60:
	AllGohomeTon[2].IN:=FALSE;
	Mach_Control.Ca_b.Ca_BeltGohomeHMI:=FALSE;
	Mach_Control.TJ_b.TJIniti_Hbtn:=FALSE;
	AllGohomeStep:=70;

70:
	AllGohomeTon[3].IN:=TRUE;
	IF AllGohomeTon[3].Q AND Mach_Control.Ca_b.Ca_BeltGohomeDone AND Mach_Control.TJ_b.TJIniti_Done THEN
	AllGohomeStep:=80;	
	END_IF	
80:
AllGohomeTon[3].IN:=FALSE;
AllGohomeStep:=888;	
END_CASE
END_ACTION

ACTION An_Alarm:


//报警时间
An_AlarmTon[1](IN:= , PT:=T#80MS , Q=> , ET=> );//正极送片搬运升降有真空信号，无极片报警延时
An_AlarmTon[2](IN:= , PT:=T#80MS , Q=> , ET=> );//正极送片搬运升降有极片，无真空信号报警延时
An_AlarmTon[3](IN:= , PT:=T#150MS , Q=> , ET=> );//正极叠台搬运升降有真空信号，无极片报警延时
An_AlarmTon[4](IN:= , PT:=T#80MS , Q=> , ET=> );//正极叠台搬运升降有极片，无真空信号报警延时
An_AlarmTon[5](IN:= , PT:=T#80MS , Q=> , ET=> );//正极纠偏平台有真空信号，无极片报警延时
An_AlarmTon[6](IN:= , PT:=T#150MS , Q=> , ET=> );//正极纠偏平台有极片，无真空信号报警延时
An_AlarmTon[7](IN:= , PT:=T#80MS , Q=> , ET=> );//正极纠偏平台连续NG
An_AlarmTon[8](IN:= , PT:=T#80MS , Q=> , ET=> );
An_AlarmTon[9](IN:= , PT:=T#300MS , Q=> , ET=> );
An_AlarmTon[10](IN:= , PT:=T#400MS , Q=> , ET=> );//
An_AlarmTon[11](IN:= , PT:=T#300MS , Q=> , ET=> );//正极极片对齐度检测返回结果超时
An_AlarmTon[12](IN:= , PT:=T#400MS , Q=> , ET=> );//正极CCD纠偏平台检测返回结果超时
An_AlarmTon[13](IN:=AnCCDMark , PT:=T#50MS , Q=> , ET=> );//正极CCD纠偏平台检测返回结果超时

An_AlarmTon[15](IN:= , PT:=T#50MS , Q=> , ET=> );//正极CCD纠偏平台检测返回结果超时
An_AlarmTon[16](IN:= , PT:=T#50MS , Q=> , ET=> );//正极CCD纠偏平台检测返回结果超时
An_AlarmTon[17](IN:=NOT Mach_Control.se.AnNGboxsensor , PT:=T#5S , Q=> , ET=> );//正极NG料盒料满

rAnUse[2](CLK:=Mach_Control.An_b.An_CCDStart AND NOT   Mach_Control.An_b.Demarcateing , Q=> );
rAnUse[3](CLK:=Par.stDT_date.An_Rectifydev_Btn , Q=> );
rAnUse[4](CLK:=arrCyCtrl[arrCyNo.ElectValveName.AnCarryingVacuum].Io.DOStatus1 , Q=> );  
rAnUse[5](CLK:= NOT arrCyCtrl[arrCyNo.ElectValveName.AnDTCarryingVacuum].Io.DOStatus1 , Q=> );

//Mach_Control.An_b.Error[1] :=TRUE;//正极送片搬运升降有真空信号，无极片报警
//Mach_Control.An_b.Error[2] :=TRUE;//正极送片搬运升降有极片，无真空信号报警
//Mach_Control.An_b.Error[3]:=TRUE;//正极叠台搬运升降在叠片过程中真空报警，请检查叠台是否掉片
//Mach_Control.An_b.Error[4] :=TRUE;//正极叠台搬运升降有极片，无真空信号报警
//Mach_Control.An_b.Error[5]:=TRUE;//正极纠偏平台有真空信号，无极片报警
//Mach_Control.An_b.Error[6]:=TRUE;//正极纠偏平台有极片，无真空信号报警
//Mach_Control.An_b.Error[7]:=TRUE;//纠偏CCD拍照完成IO信号未给出
//Mach_Control.An_b.Error[8]  ;//CCD标定NG
//Mach_Control.An_b.Error[9]  ;
//Mach_Control.An_b.Error[10]  ;
//Mach_Control.An_b.Error[11]:=TRUE;//正极有凸轮耦合报警
//Mach_Control.An_b.Error[12]:=TRUE;//正极NG收纳盒满料报警
//Mach_Control.An_b.Error[13];
//Mach_Control.An_b.Error[14]:=TRUE;//正极防撞感应信号报警
//Mach_Control.An_b.Error[15]
//Mach_Control.An_b.Error[16]
//Mach_Control.An_b.Error[17]
//Mach_Control.An_b.Error[18] :=TRUE;//正极CCD纠偏平台检测返回结果超时
// Mach_Control.An_b.Error[19]:=TRUE;//正极回原点超时报警
// Mach_Control.An_b.Error[20];
//Mach_Control.An_b.Error[21]:=TRUE;//正极纠偏平台连续NG
//Mach_Control.An_b.Error[22]:=TRUE;//正极叠台搬运升降真空报警，电芯上有片，请拿掉
//Mach_Control.An_b.Error[23]:=TRUE;//正极叠台搬运升降真空报警，电芯上无掉片
//Mach_Control.An_b.Error[24] ////正极纠偏平台NG片未排掉报警，请拿掉
//Mach_Control.An_b.Error[25] ////正极极片对齐度检测返回结果超时
//Mach_Control.An_b.Error[26] ////正极搬运防撞软限位报警
//Mach_Control.An_b.Error[27]//    //正极极片对齐度检测返回结果无片报警
//Mach_Control.An_b.Error[28]//正极叠片完空叠隔膜时，正极叠片搬运机械手真空有信号、标记有极片报警,请拿掉极片
//Mach_Control.An_b.Error[29]:=TRUE;		//正极初始化时正极叠片搬运升降吸盘有真空报警
//Mach_Control.An_b.Error[30]:=TRUE;		//正极初始化时正极送片搬运升降吸盘有真空报警	

//Mach_Control.An_b.Error[32]:=TRUE;//正极送片搬运在叠片过程中真空报警
//Mach_Control.An_b.Error[33]:=FALSE;//纠偏平台有片，请拿走
//Mach_Control.An_b.Error[34]:=FALSE;//正极叠台搬运平移取片时真空报警,请确认纠偏台是否掉片
//Mach_Control.An_b.Error[35]:=TRUE;//正极纠偏台NG料盒料满报警
//Mach_Control.An_b.Error[36]:=TRUE;//正极纠偏纠偏CCD返回结果超时
//Mach_Control.An_b.Error[37]:=TRUE;//正极叠台搬运升降有真空信号，无极片报警
//Mach_Control.An_b.Error[38] :=TRUE;//正极叠台搬运升降有极耳无真空报警
//Mach_Control.An_b.Error[39] :=TRUE;//正极叠台搬运升降有极耳无真空报警
//Mach_Control.An_b.Error[40] S=AnOverNGcount>=3;//正极单张踢废连续NG
//Mach_Control.An_b.Error[41] :=TRUE;//正极机械手初始化时，叠台搬运升降不在避让位
Mach_Control.An_b.Error[40] S=AnOverNGcount>=3;//正极单张踢废连续NG

//NG料盒料满报警
	IF (*Par.stDT_date.An_Rectifydev_JS>=Par.stDT_date.An_Rectifydev_NGSet OR*) An_AlarmTon[17].Q THEN
		Mach_Control.An_b.Error[35]:=TRUE;//负极纠偏台NG料盒料满报警
	ELSE
		Mach_Control.An_b.Error[35]:=FALSE;//负极纠偏台NG料盒料满报警
	END_IF
	IF rAnUse[3].Q THEN
		Par.stDT_date.An_Rectifydev_JS:=0;
	END_IF



//正极初始化时有真空报警	
	IF Mach_Control.An_b.An_GohomeHMI THEN
		IF arrCyCtrl[arrCyNo.ElectValveName.AnDTCarryingVacuum].Status.ONState  THEN    
			Mach_Control.An_b.Error[29]:=TRUE;		//正极初始化时正极叠片搬运升降吸盘有真空报警
		END_IF
		IF arrCyCtrl[arrCyNo.ElectValveName.	AnCarryingVacuum	].Status.ONState THEN	
			Mach_Control.An_b.Error[30]:=TRUE;		//正极初始化时正极送片搬运升降吸盘有真空报警	
		END_IF		 
	END_IF	
(*
//正极送片搬运升降真空信号与有无极片标记不一致报警
An_AlarmTon[1].IN:=arrCyCtrl[arrCyNo.ElectValveName.AnCarryingVacuum].Io.DIOnSwitch AND NOT Mach_Control.An_b.An_CarryingFalg 
	AND NOT Mach_Control.U.EmptyRunMode AND NOT Mach_Control.An_b.Error[2]  AND NOT Blueflaging AND Mach_Control.U.DT_iMode=1;
		IF  An_AlarmTon[1].Q THEN
				Mach_Control.An_b.Error[1] :=TRUE;//正极送片搬运升降有真空信号，无极片报警
		END_IF
*)
//正极送片搬运升降有极片，无真空信号报警------取片过程中真空报警判断
An_AlarmTon[2].IN:=NOT arrCyCtrl[arrCyNo.ElectValveName.AnCarryingVacuum].Io.DIOnSwitch AND  Mach_Control.An_b.An_CarryingFalg  AND
	 arrAxisCtrl[AxiseNo.AxisName.AnCarryingUpDown].Status.fActPos<=(arrAxisPar[AxiseNo.AxisName.AnCarryingUpDown].arrTargetPoint[2]-5) 
	AND arrAxisCtrl[AxiseNo.AxisName.AnCarryingLine].Status.NoMoving AND NOT Mach_Control.U.EmptyRunMode ;
	IF  An_AlarmTon[2].Q THEN
			Mach_Control.An_b.Error[2] :=TRUE;//正极送片搬运升降有极片，无真空信号报警
			(*
			Mach_Control.An_b.An_CarryingFalg:=FALSE;
			arrCyCtrl[arrCyNo.ElectValveName.AnCarryingVacuum].Cmd.bOFF:=TRUE;//正极搬运升降取料真空关
			arrCyCtrl[arrCyNo.ElectValveName.AnCarryingVacuum].Cmd.bON:=FALSE;//正极搬运升降取料真空关
			arrCyCtrl[arrCyNo.ElectValveName.AnCarryingVacuumBark].Cmd.bON:=TRUE;//正极搬运升降取料破真空开
			arrCyCtrl[arrCyNo.ElectValveName.AnCarryingVacuumBark].Cmd.bOFF:=FALSE;//正极搬运升降取料破真空开
			*)
	END_IF
IF 	Mach_Control.An_b.Error[2]AND arrCyCtrl[arrCyNo.ElectValveName.AnCarryingVacuum].Io.DIOnSwitch AND  rAn_AlarmRest.Q  THEN
	Mach_Control.An_b.Error[2] :=FALSE;//正极送片搬运升降有极片，无真空信号报警
ELSIF Mach_Control.An_b.Error[2]AND NOT arrCyCtrl[arrCyNo.ElectValveName.AnCarryingVacuum].Io.DIOnSwitch AND  rAn_AlarmRest.Q  THEN
	arrCyCtrl[arrCyNo.ElectValveName.AnCarryingVacuum].Cmd.bOFF:=TRUE;//正极搬运升降取料真空关
	arrCyCtrl[arrCyNo.ElectValveName.AnCarryingVacuum].Cmd.bON:=FALSE;//正极搬运升降取料真空关
	arrCyCtrl[arrCyNo.ElectValveName.AnCarryingVacuumBark].Cmd.bON:=TRUE;//正极搬运升降取料破真空开
	arrCyCtrl[arrCyNo.ElectValveName.AnCarryingVacuumBark].Cmd.bOFF:=FALSE;//正极搬运升降取料破真空开
	An_StandbyStep1:=0;
	An_Step0:=0;
	An_Step1:=0;
	An_Step2:=0;
	An_Step3:=0;
	Mach_Control.An_b.Error[2] :=FALSE;//正极送片搬运升降有极片，无真空信号报警
	Mach_Control.An_b.An_CarryingFalg:=FALSE;
END_IF
	
	
	
	
	
//正极送片搬运在叠片过程中的真空信号判断
	An_AlarmTon[15].IN:=NOT arrCyCtrl[arrCyNo.ElectValveName.AnCarryingVacuum].Io.DIOnSwitch AND  Mach_Control.An_b.An_CarryingFalg 
	AND NOT Mach_Control.U.EmptyRunMode AND arrAxisCtrl[AxiseNo.AxisName.AnCarryingLine].Status.Moving	  
	 AND  arrAxisCtrl[AxiseNo.VirAxisName.VirMain].Status.fActPos<232 AND  arrAxisCtrl[AxiseNo.VirAxisName.VirMain].Status.fActPos>1   ;
	IF  An_AlarmTon[15].Q THEN
		CCD.AnRec.Finish.RectifyResult:=0;
		Mach_Control.An_b.Error[32] :=TRUE;//正极送片搬运升降有极片，无真空信号报警
		Mach_Control.An_b.An_CarryingFalg:=FALSE;
		arrCyCtrl[arrCyNo.ElectValveName.AnCarryingVacuum].Cmd.bOFF:=TRUE;//正极搬运升降取料真空关
		arrCyCtrl[arrCyNo.ElectValveName.AnCarryingVacuum].Cmd.bON:=FALSE;//正极搬运升降取料真空关
		arrCyCtrl[arrCyNo.ElectValveName.AnCarryingVacuumBark].Cmd.bON:=TRUE;//正极搬运升降取料破真空开
		arrCyCtrl[arrCyNo.ElectValveName.AnCarryingVacuumBark].Cmd.bOFF:=FALSE;//正极搬运升降取料破真空开
	END_IF
	IF Mach_Control.An_b.Error[32] AND rAn_AlarmRest.Q   THEN
		//CCD.AnRec.Finish.RectifyResult:=0;
		CCD.AnRec.Start.iPhotoDo:=1;//第二次拍照
		Mach_Control.An_b.An_CCDStart :=TRUE;//启动CCD拍照
	END_IF
	IF Mach_Control.An_b.Error[32] AND (CCD.AnRec.Finish.RectifyResult=3  OR  Mach_Control.U.CCD_ChosesHMI) AND rAn_AlarmRest.Q  THEN
		Mach_Control.An_b.Error[32]:=FALSE;
		Mach_Control.An_b.Error[33]:=FALSE;//纠偏平台有片，请拿走
	END_IF
	IF Mach_Control.An_b.Error[32] AND (CCD.AnRec.Finish.RectifyResult<>3  AND NOT   Mach_Control.U.CCD_ChosesHMI)THEN
		Mach_Control.An_b.Error[33]:=TRUE;//纠偏平台有片，请拿走
	END_IF
	
	
	
	
	
//正极叠片搬运升降真空信号与有无极片标记不一致报警
An_AlarmTon[3].IN:=(arrCyCtrl[arrCyNo.ElectValveName.AnDTCarryingVacuum].Io.DIOnSwitch OR Mach_Control.se.AnDTCarryingJROnSwitch)
    AND NOT Mach_Control.An_b.An_DPCarryingFalg AND Mach_Control.U.DT_iMode=1 
	AND NOT Mach_Control.U.EmptyRunMode AND (An_Step2=0 OR An_Step2=6666) AND NOT Mach_Control.An_b.Error[4] AND iEmptyFoldStep[1]=0 
	AND arrAxisCtrl[AxiseNo.AxisName.AnDTCarryingUpDown].Status.fActPos<=(arrAxisPar[AxiseNo.AxisName.AnDTCarryingUpDown].arrTargetPoint[2]-5)  
	AND DP_Step0<1000 AND DP_Step0>3100;
	IF  An_AlarmTon[3].Q THEN
		IF arrCyCtrl[arrCyNo.ElectValveName.AnDTCarryingVacuum].Io.DIOnSwitch THEN
			Mach_Control.An_b.Error[3]:=TRUE;//正极叠台搬运升降有真空信号，无极片报警
		END_IF
        IF 	Mach_Control.se.AnDTCarryingJROnSwitch THEN
			Mach_Control.An_b.Error[37]:=TRUE;//正极叠台搬运升降有真空信号，无极片报警
		END_IF
	END_IF

	
//正极叠台搬运升降有极片，无真空信号报警-------叠片搬运平移取片过程真空检测
An_AlarmTon[16].IN:=(NOT arrCyCtrl[arrCyNo.ElectValveName.AnDTCarryingVacuum].Io.DIOnSwitch OR NOT Mach_Control.se.AnDTCarryingJROnSwitch)
     AND  Mach_Control.An_b.An_DPCarryingFalg  AND (An_Step2=0 OR An_Step2=6666) AND
	arrAxisCtrl[AxiseNo.AxisName.AnDTCarryingUpDown].Status.fActPos<=(arrAxisPar[AxiseNo.AxisName.AnDTCarryingUpDown].arrTargetPoint[2]-5)  
	AND  arrAxisCtrl[AxiseNo.AxisName.AnDTCarryingLine].Status.NoMoving AND NOT Mach_Control.U.EmptyRunMode AND iEmptyFoldStep[1]=0 
	AND (DP_Step0<1000 OR DP_Step0>3100)  ;//
	IF  An_AlarmTon[16].Q THEN
		//CCD.AnRec.Finish.RectifyResult:=0;//拍照结果清零
		IF NOT arrCyCtrl[arrCyNo.ElectValveName.AnDTCarryingVacuum].Io.DIOnSwitch THEN
		   Mach_Control.An_b.Error[34] :=TRUE;//正极叠台搬运升降有极片，无真空信号报警
		END_IF  
		IF NOT Mach_Control.se.AnDTCarryingJROnSwitch THEN
           Mach_Control.An_b.Error[39] :=TRUE;//正极叠台搬运升降有极耳无真空报警
        END_IF   
		Mach_Control.An_b.An_DPCarryingFalg:=FALSE;
		arrCyCtrl[arrCyNo.ElectValveName.AnDTCarryingVacuum].Cmd.bOFF:=FALSE;//正极叠片搬运升降真空关
		arrCyCtrl[arrCyNo.ElectValveName.AnDTCarryingVacuum].Cmd.bON:=TRUE;//正极叠片搬运升降真空关
		//arrCyCtrl[arrCyNo.ElectValveName.AnDTCarryingVacuumBark].Cmd.bON:=TRUE;//正极叠片搬运破真空开
		//arrCyCtrl[arrCyNo.ElectValveName.AnDTCarryingVacuumBark].Cmd.bOFF:=FALSE;//正极叠片搬运破真空关
	END_IF
//叠台搬运平移在取片过程中报警时，纠偏平台拍照有无片来确定是否掉片到纠偏平台
	IF (Mach_Control.An_b.Error[34] OR Mach_Control.An_b.Error[39]) AND rAn_AlarmRest.Q  THEN
		//CCD.AnRec.Finish.RectifyResult:=0;//拍照结果清零
		Mach_Control.An_b.An_CCDStart :=TRUE;//启动CCD拍照
		CCD.AnRec.Start.iPhotoDo:=1;//启动CCD第二次拍照
	END_IF
	IF (Mach_Control.An_b.Error[34] OR Mach_Control.An_b.Error[39]) AND (CCD.AnRec.Finish.RectifyResult=3  OR  Mach_Control.U.CCD_ChosesHMI) AND rAn_AlarmRest.Q  THEN
		Mach_Control.An_b.Error[34]:=FALSE;//叠台升降取片过程中真空报警，
		Mach_Control.An_b.Error[39]:=FALSE;//叠台升降取片过程中真空报警，
		Mach_Control.An_b.Error[33]:=FALSE;//纠偏平台有片，请拿走
	ELSIF( Mach_Control.An_b.Error[34] OR Mach_Control.An_b.Error[39]) AND (CCD.AnRec.Finish.RectifyResult<>3  AND NOT   Mach_Control.U.CCD_ChosesHMI)THEN
		Mach_Control.An_b.Error[33]:=TRUE;//纠偏平台有片，请拿走
	END_IF
	






	
	
//正极叠台搬运升降有极片，无真空信号报警-------叠片搬运平移叠片过程真空检测
An_AlarmTon[4].IN:=(NOT arrCyCtrl[arrCyNo.ElectValveName.AnDTCarryingVacuum].Io.DIOnSwitch OR NOT Mach_Control.se.AnDTCarryingJROnSwitch)
     AND  Mach_Control.An_b.An_DPCarryingFalg  AND (An_Step2=0 OR An_Step2=6666) AND
	 arrAxisCtrl[AxiseNo.VirAxisName.VirMain].Status.fActPos<232 AND  arrAxisCtrl[AxiseNo.VirAxisName.VirMain].Status.fActPos>1  AND NOT Mach_Control.U.EmptyRunMode
	AND  arrAxisCtrl[AxiseNo.AxisName.AnDTCarryingLine].Status.Moving	 ;//
	IF  An_AlarmTon[4].Q THEN
		//Mach_Control.DT_b.OverhandResult:=0;
		IF NOT arrCyCtrl[arrCyNo.ElectValveName.AnDTCarryingVacuum].Io.DIOnSwitch THEN
		  Mach_Control.An_b.Error[4] :=TRUE;//正极叠台搬运升降有极片，无真空信号报警
	    END_IF
		IF  NOT Mach_Control.se.AnDTCarryingJROnSwitch THEN
		  Mach_Control.An_b.Error[38] :=TRUE;//正极叠台搬运升降有极耳无真空报警
		END_IF
		An_Number:=TRUE;
		Mach_Control.An_b.An_DPCarryingFalg:=FALSE;
		arrCyCtrl[arrCyNo.ElectValveName.AnDTCarryingVacuum].Cmd.bOFF:=FALSE;//正极叠片搬运升降真空关
		arrCyCtrl[arrCyNo.ElectValveName.AnDTCarryingVacuum].Cmd.bON:=TRUE;//正极叠片搬运升降真空关
		//arrCyCtrl[arrCyNo.ElectValveName.AnDTCarryingVacuumBark].Cmd.bON:=TRUE;//正极叠片搬运破真空开
		//arrCyCtrl[arrCyNo.ElectValveName.AnDTCarryingVacuumBark].Cmd.bOFF:=FALSE;//正极叠片搬运破真空关
	END_IF
	
	//正极叠台搬运升降真空报警，电芯上有片，请拿掉
	An_AlarmTon[8].IN:=(Mach_Control.An_b.Error[4] OR Mach_Control.An_b.Error[38]) AND Mach_Control.DT_b.OverhandResult<>3 AND NOT Mach_Control.U.CCD_ChosesHMI ;
	IF  An_AlarmTon[8].Q THEN
		Mach_Control.An_b.Error[22]:=TRUE;//正极叠台搬运升降真空报警，电芯上有片，请拿掉
	END_IF
	IF fAn_AlarmRest.Q AND  Mach_Control.An_b.Error[22] AND arrAxisCtrl[AxiseNo.VirAxisName.VirMain].Status.fActPos<1  THEN
		Mach_Control.DT_b.OverhandResult:=0;
		CCD.Over.Start.iPhotoDo:=2;
		Mach_Control.DT_b.CDD_OverStart:=TRUE;
	END_IF

	IF Mach_Control.An_b.Error[22] AND Mach_Control.DT_b.OverhandResult=3  AND rAn_AlarmRest.Q THEN
		Mach_Control.An_b.Error[22]:=FALSE;//复位电芯有片报警
		Mach_Control.DT_b.OverhandResult:=0;
	END_IF
	
	//正极叠台搬运升降真空报警，电芯上无掉片
	An_AlarmTon[9].IN:=(Mach_Control.An_b.Error[4] OR Mach_Control.An_b.Error[38] )AND Mach_Control.DT_b.OverhandResult=3 AND NOT Mach_Control.U.CCD_ChosesHMI ;
	IF  An_AlarmTon[9].Q THEN
		Mach_Control.An_b.Error[23]:=TRUE;//正极叠台搬运升降真空报警，电芯上无掉片
	END_IF

	
	

//正极纠偏平台真空信号与有无极片标记不一致报警
An_AlarmTon[5].IN:=arrCyCtrl[arrCyNo.ElectValveName.AndeviationVacuum].Io.DIOnSwitch AND NOT Mach_Control.An_b.An_deviationFalg 
	AND NOT Mach_Control.U.EmptyRunMode AND arrAxisCtrl[AxiseNo.AxisName.AnDTCarryingUpDown].Status.Homed 
	AND arrAxisCtrl[AxiseNo.AxisName.AnDTCarryingUpDown].Status.fActPos<=(arrAxisPar[AxiseNo.AxisName.AnDTCarryingUpDown].arrTargetPoint[4]+5) 
	AND iEmptyFoldStep[1]=0 AND (DP_Step0<1000 OR DP_Step0>3100) ;
	IF  An_AlarmTon[5].Q THEN
		Mach_Control.An_b.Error[5]:=TRUE;//正极纠偏平台有真空信号，无极片报警
	END_IF

//正极纠偏平台有极片，无真空信号报警
An_AlarmTon[6].IN:=NOT arrCyCtrl[arrCyNo.ElectValveName.AndeviationVacuum].Io.DIOnSwitch AND Mach_Control.An_b.An_deviationFalg 
	AND NOT Mach_Control.U.EmptyRunMode AND	arrAxisCtrl[AxiseNo.AxisName.AnCarryingUpDown].Status.Homed  
	AND arrAxisCtrl[AxiseNo.AxisName.AnCarryingUpDown].Status.fActPos<=(arrAxisPar[AxiseNo.AxisName.AnCarryingUpDown].arrTargetPoint[4]+5) 
	AND iEmptyFoldStep[1]=0 AND (DP_Step0<1000 OR DP_Step0>3100) AND NOT Mach_Control.An_b.An_VacuumErrorNG ;
	IF An_AlarmTon[6].Q  THEN
		Mach_Control.An_b.Error[6]:=TRUE;//正极纠偏平台有极片，无真空信号报警
		Mach_Control.An_b.An_VacuumErrorNG:=TRUE;//正极抛真空NG料标志
	END_IF

//正极纠偏平台连续NG
An_AlarmTon[7].IN:=Mach_Control.An_b.An_CCD_amount>=3 AND NOT Mach_Control.An_b.Error[21] AND NOT Mach_Control.U.CCD_ChosesHMI ;
	IF  An_AlarmTon[7].Q THEN
			Mach_Control.An_b.Error[21]:=TRUE;//正极纠偏平台连续NG
	END_IF	
//
IF Mach_Control.An_b.Error[24] AND CCD.AnRec.Finish.RectifyResult=3  AND rAn_AlarmRest.Q THEN
	Mach_Control.An_b.Error[24]:=FALSE;
END_IF
IF fAn_AlarmRest.Q AND Mach_Control.An_b.Error[24] AND arrAxisCtrl[AxiseNo.VirAxisName.VirMain].Status.fActPos<1  THEN	
	CCD.AnRec.Start.iPhotoDo:=1;//第二次拍照
	Mach_Control.An_b.An_CCDStart :=TRUE;//启动CCD拍照
END_IF

//正极取片报警复位
rAn_AlarmRest(CLK:=Sys_Control.btn.System_Rrestbtn , Q=> );//正极报警复位上升沿
fAn_AlarmRest(CLK:=Sys_Control.btn.System_Rrestbtn , Q=> );//正极报警复位下降沿
IF Mach_Control.U.DT_iMode=3 THEN//在手动状态下，复位报警
	
		//IF Mach_Control.An_b.Error[2] AND rAn_AlarmRest.Q THEN
				//Mach_Control.An_b.An_CarryingFalg :=FALSE;
		//END_IF
		
		IF (Mach_Control.An_b.Error[4] OR Mach_Control.An_b.Error[38]) AND rAn_AlarmRest.Q THEN
				Mach_Control.An_b.An_DPCarryingFalg:=FALSE;
		END_IF
//20240105临时屏蔽	
(*		IF Mach_Control.An_b.Error[6] AND rAn_AlarmRest.Q  THEN
				Mach_Control.An_b.An_deviationFalg :=FALSE;
		END_IF
*)		
		IF Mach_Control.An_b.Error[21] AND rAn_AlarmRest.Q  THEN
				Mach_Control.An_b.An_CCD_amount:=0;
		END_IF
																		//20240105临时屏蔽	
		IF ((Mach_Control.An_b.Error[2] AND NOT Mach_Control.An_b.An_CarryingFalg)OR Mach_Control.An_b.Error[4] OR Mach_Control.An_b.Error[38] (*OR Mach_Control.An_b.Error[6]*)) AND rAn_AlarmRest.Q  THEN
				An_StandbyStep1:=0;
				An_Step0:=0;
				An_Step1:=0;
				An_Step2:=0;
				An_Step3:=0;
		END_IF
		
		IF fAn_AlarmRest.Q AND NOT Mach_Control.An_b.Error[22]  AND NOT Mach_Control.An_b.Error[2] 
			AND NOT Mach_Control.An_b.Error[4] AND NOT Mach_Control.An_b.Error[24] 
			AND NOT Mach_Control.An_b.Error[32]  AND NOT Mach_Control.An_b.Error[34]
            AND NOT Mach_Control.An_b.Error[38] AND NOT Mach_Control.An_b.Error[39] THEN
				MEMSET(ADR(Mach_Control.An_b.Error),0,SIZEOF(Mach_Control.An_b.Error)); // 正极取片报警复位	
				//AnOverNGcount:=0;
				arrAxisCtrl[AxiseNo.AxisName.AnDTCarryingLine].Cmd.bStop:=FALSE;
		END_IF		
	
			IF AnOverNGcount>= 3 AND fAn_AlarmRest.Q THEN
		    	AnOverNGcount:=0;
		   END_IF	
		
		IF Mach_Control.An_b.An_DTqr AND Mach_Control.An_b.Error[2] THEN
			 	Mach_Control.An_b.Error[2] :=FALSE;
				Mach_Control.An_b.An_CarryingFalg :=FALSE;
		END_IF
		
		IF Mach_Control.An_b.An_DTqr AND  (Mach_Control.An_b.Error[4] OR Mach_Control.An_b.Error[38]) THEN
			 	Mach_Control.An_b.Error[4] :=FALSE;
				Mach_Control.An_b.Error[38] :=FALSE;
				Mach_Control.An_b.An_DPCarryingFalg:=FALSE;
		END_IF
		
		IF (Mach_Control.An_b.Error[7] OR An_StandbyStep0=9999) AND fAn_AlarmRest.Q THEN
				Mach_Control.An_b.Error[7] :=FALSE;
				An_StandbyStep0:=0;
		END_IF
		
		IF fAn_AlarmRest.Q THEN
				IF 9991<=An_StandbyStep1 AND An_StandbyStep1<=10000 THEN
						An_StandbyStep1:=1000;
						An_Step0:=0;
						An_Step1:=0;
						An_Step2:=0;
						An_Step3:=0;
				END_IF
		END_IF
END_IF

     An_dppy_Xzb:=arrAxisPar[AxiseNo.AxisName.AnCarryingLine].arrTargetPoint[2]+arrAxisCtrl[AxiseNo.AxisName.AnDTCarryingLine].Status.fActPos;

    IF An_Step3=30 AND NOT arrAxis[AxiseNo.AxisName.AnDTCarryingLine].Status.Coupled AND  NOT arrAxis[AxiseNo.AxisName.AnCarryingLine].Status.Coupled   AND   arrAxis[AxiseNo.VirAxisName.VirMain].Status.NotMoving 
		  AND arrAxisCtrl[AxiseNo.AxisName.AnCarryingLine].Status.Homed AND arrAxisCtrl[AxiseNo.AxisName.AnDTCarryingLine].Status.Homed AND NOT  arrAxisCtrl[AxiseNo.AxisName.AnCarryingLine].Cmd.arrbRealPoint[1]
          AND ABS((arrAxisPar[AxiseNo.AxisName.AnCarryingLine].arrTargetPoint[2]+arrAxisCtrl[AxiseNo.AxisName.AnDTCarryingLine].Status.fActPos)-arrAxisCtrl[AxiseNo.AxisName.AnCarryingLine].Status.fActPos)
            <(ABS(arrAxisPar[AxiseNo.AxisName.AnCarryingLine].arrTargetPoint[2]-arrAxisPar[AxiseNo.AxisName.AnCarryingLine].arrTargetPoint[1])+arrAxisPar[AxiseNo.AxisName.AnDTCarryingLine].arrTargetPoint[1]-20) THEN
	   Mach_Control.An_b.Error[26]:=TRUE;//正极搬运防撞软限位报警
	END_IF
	
	AnError_r(CLK:= Mach_Control.An_b.Error[26] , Q=> );
	IF AnError_r.Q THEN 
	   arrAxisCtrl[AxiseNo.AxisName.AnCarryingLine].Cmd.bStop:=TRUE;
       arrAxisCtrl[AxiseNo.AxisName.AnDTCarryingLine].Cmd.bStop :=TRUE;
	 END_IF
	 
	IF  P2M2_sysControl.btn.System_Rrestbtn THEN
			arrAxisCtrl[AxiseNo.AxisName.AnCarryingLine].Cmd.bStop:=FALSE;
			arrAxisCtrl[AxiseNo.AxisName.AnDTCarryingLine].Cmd.bStop :=FALSE;
	END_IF

	
//空叠隔膜时检查叠台升降有没有片
IF Mach_Control.U.DT_iMode=3 THEN//在手动状态下，复位报警	
		IF  Mach_Control.An_b.Error[28] AND DP_Step0=2070 AND rAn_AlarmRest.Q  THEN
				Mach_Control.An_b.An_DPCarryingFalg:=FALSE;
		END_IF
END_IF

//ccdJ拍照检测返回结果超时报警
rAnCCDStart(CLK:=Mach_Control.An_b.An_CCDStart , Q=> );
IF rAnCCDStart.Q THEN
  	 AnCCDMark:=TRUE;
END_IF
 
IF AnCCDMark AND CCD.AnRec.Finish.RectifyResult=0  AND NOT Mach_Control.U.CCD_ChosesHMI THEN
		IF NOT An_AlarmTon[12].Q THEN
			An_AlarmTon[12].IN:=TRUE;
		ELSE
			Mach_Control.An_b.Error[18] :=TRUE;//正极CCD纠偏平台检测返回结果超时
			AnCCDMark :=FALSE;
		END_IF
ELSE
		An_AlarmTon[12].IN:=FALSE;
END_IF

IF (Mach_Control.An_b.Error[18] AND Sys_Control.btn.System_Rrestbtn) OR
	   (CCD.AnRec.Finish.RectifyResult<>0 AND  AnCCDMark  AND An_AlarmTon[13].Q  ) THEN
	   AnCCDMark :=FALSE;
	   An_AlarmTon[12].IN:=FALSE;
END_IF

IF Mach_Control.U.DT_iMode=1 AND  rAnUse[4].Q THEN
 Par.stDT_date.An_sucker1_JS :=Par.stDT_date.An_sucker1_JS+1;
END_IF

IF( HMI_Hour>=7  AND HMI_Hour<9) OR (HMI_Hour>=19  AND HMI_Hour<21) THEN
      IF Par.stDT_date.An_sucker1_JS>=Par.stDT_date.An_sucker1Set THEN
	      Mach_Control.An_b.Error[42]:=TRUE;//正极送片搬运吸盘计数到达设定值
      END_IF
END_IF
IF Mach_Control.DT_b.An_sucker1_JSclear THEN
   Par.stDT_date.An_sucker1_JS:=0;
END_IF  

IF Mach_Control.U.DT_iMode=1 AND  rAnUse[5].Q THEN
 Par.stDT_date.An_sucker2_JS  :=Par.stDT_date.An_sucker2_JS +1;
END_IF

IF( HMI_Hour>=7  AND HMI_Hour<9) OR (HMI_Hour>=19  AND HMI_Hour<21) THEN
      IF Par.stDT_date.An_sucker2_JS >=Par.stDT_date.An_sucker2Set  THEN
	      Mach_Control.An_b.Error[43]:=TRUE;//正极叠台搬运吸盘计数到达设定值
      END_IF
END_IF
IF Mach_Control.DT_b.An_sucker2_JSclear THEN
   Par.stDT_date.An_sucker2_JS:=0;
END_IF  
(*
IF An_CCDNG>=10 THEN
		Mach_Control.An_b.Error[12]:=TRUE;//正极NG收纳盒满料报警
END_IF

IF Mach_Control.An_b.Error[12] AND P2M2_sysControl.btn.System_Rrestbtn THEN
		 Mach_Control.An_b.Error[12]:=FALSE;
		 An_CCDNG:=0;
END_IF

*)
END_ACTION

ACTION An_Cam:
An_Cam_ton[1](PT:=T#100MS);
An_Cam_ton[2](PT:=T#100MS);
An_Cam_ton[3](PT:=T#100MS);
An_Cam_ton[4](PT:=T#100MS);
An_Cam_ton[5](PT:=T#100MS);

(***********************************正极凸轮表创建************************************************)
(*
     fbCrectCamLeftYDLine                   :FB_CrectCamYaDaoLine ;
     fbCrectCamLeftYDUpDown             :FB_CrectCamYaDaoUpDown ;
     fbCrectCamRightYDLine                 :FB_CrectCamYaDaoLine ;
     fbCrectCamRightYDUpDown           :FB_CrectCamYaDaoUpDown ;
*)
//正极送纠偏搬运平移凸轮创建
fbAnCrectCamCarryingLine.fMoveLength:=ABS(arrAxisPar[AxiseNo.AxisName.AnCarryingLine].arrTargetPoint[1]-arrAxisPar[AxiseNo.AxisName.AnCarryingLine].arrTargetPoint[2]);
fbAnCrectCamCarryingLine(
	bCreatTable:=                fbAnCrectCamCarryingLine.bCreatTable , 
	Reset:=                          stSysState.bReset  ,  
	iTable:=                       TableNo.M_AnCarryingLine  , 
	fMoveLength:=              , 
	fMasterKeyPos:=          250 , //
	
	axisMaster:=                 arrAxis[AxiseNo.VirAxisName.VirMain] ,  
    axisSlave:=                    arrAxis[AxiseNo.AxisName.AnCarryingLine] ,  
	bCreatTableDone=> , 
	bCreatTableError=> , 
	bError=> );

fbAnCrectCamCarryingLine.bCreatTableDone;
fbAnCrectCamCarryingLine.bCreatTableError;
fbAnCrectCamCarryingLine.bError;
//正极送纠偏搬运升降取片凸轮创建
(*
fbAnCrectCamCarryingUpDown(
	bCreatTable:=fbAnCrectCamCarryingUpDown.bCreatTable, 
	Reset:=stSysState.bReset  , 
	iTable:=TableNo.M_AnCarryingUpDown , 
	fMoveLength:=arrAxisPar[AxiseNo.AxisName.AnCarryingUpDown].arrTargetPoint[2], //取片高度
	fSaveLength:=arrAxisPar[AxiseNo.AxisName.AnCarryingUpDown].arrTargetPoint[1] , //安全高度
	fInitLength:=arrAxisPar[AxiseNo.AxisName.AnCarryingUpDown].arrTargetPoint[4],//升降轴耦合初始位
	fMasterKeyPos1:=90 , //72
	fMasterKeyPos2:=180 , //144
	fMasterKeyPos3:=229 , //198
	fMasterKeyPos4:=310 , //324
	axisSlave:=arrAxis[AxiseNo.AxisName.AnCarryingUpDown]  , 
	axisMaster:=arrAxis[AxiseNo.VirAxisName.VirMain]  , 
	bCreatTableDone=> , 
	bCreatTableError=> , 
	bError=> );
	
fbAnCrectCamCarryingUpDown.bCreatTableDone;
fbAnCrectCamCarryingUpDown.bCreatTableError;
fbAnCrectCamCarryingUpDown.bError;
*)


fbAnCrectCamUpDown_4(//无用
	bCreatTable:=fbAnCrectCamUpDown_4.bCreatTable , 
	Reset:=fbAnCrectCamUpDown_4.Reset , 
	iTable:=TableNo.M_AnCarryingUpDown  , 
	fInitLength:=arrAxisPar[AxiseNo.AxisName.AnCarryingUpDown].arrTargetPoint[2], //取片高度 
	fMoveLength:=arrAxisPar[AxiseNo.AxisName.AnCarryingUpDown].arrTargetPoint[1] , //安全高度
	fSaveLength:=arrAxisPar[AxiseNo.AxisName.AnCarryingUpDown].arrTargetPoint[4],//升降轴耦合初始位
	fMasterKeyPos1:=90 , 
	fMasterKeyPos2:=180 , 
	axisSlave:=arrAxis[AxiseNo.AxisName.AnCarryingUpDown] , 
	axisMaster:=arrAxis[AxiseNo.VirAxisName.VirMain] , 
	bCreatTableDone=> , 
	bCreatTableError=> , 
	bError=> );

fbAnCrectCamUpDown_4.bCreatTableDone;
fbAnCrectCamUpDown_4.bCreatTableError;
fbAnCrectCamUpDown_4.bError;


(**********20240528SJ***************)
arrAxisPar[AxiseNo.AxisName.AnCarryingUpDown].arrTargetPoint[10]:=8; //等待高度  参数可调
arrAxisPar[AxiseNo.AxisName.AnCarryingUpDown].arrTargetPoint[11]:=18; //安全高度  参数可调
arrAxisPar[AxiseNo.AxisName.AnCarryingUpDown].arrTargetPoint[4]:=arrAxisPar[AxiseNo.AxisName.AnCarryingUpDown].arrTargetPoint[3]-arrAxisPar[AxiseNo.AxisName.AnCarryingUpDown].arrTargetPoint[10];  //等待位置
//arrAxisPar[AxiseNo.AxisName.AnCarryingUpDown].arrTargetPoint[1]:=arrAxisPar[AxiseNo.AxisName.AnCarryingUpDown].arrTargetPoint[3]-arrAxisPar[AxiseNo.AxisName.AnCarryingUpDown].arrTargetPoint[11];  //安全位置

//正极送纠偏搬运升降放片凸轮创建
fbAnCrectCamCarryingUpDown1(  //放片
	bCreatTable:=fbAnCrectCamCarryingUpDown1.bCreatTable, 
	Reset:=stSysState.bReset  , 
	iTable:=TableNo.M_AnCarryingUpDown1 , 
	fMoveLength:=    arrAxisPar[AxiseNo.AxisName.AnCarryingUpDown].arrTargetPoint[10]            , //放片高度
	fSaveLength:=    arrAxisPar[AxiseNo.AxisName.AnCarryingUpDown].arrTargetPoint[10]-arrAxisPar[AxiseNo.AxisName.AnCarryingUpDown].arrTargetPoint[11] , //安全抬升高度
	//fInitLength:=arrAxisPar[AxiseNo.AxisName.AnCarryingUpDown].arrTargetPoint[4] ,//升降轴耦合初始位
	fMasterKeyPos1:=125 , //
	fMasterKeyPos2:=250 , //
	fMasterKeyPos3:=260 , //
	fMasterKeyPos4:=320 , //
	fMasterKeyPos5:=359 , //
	//fMasterKeyPos6:=250 , //
	fSlaveVelo:=0.25 , //
	
	axisSlave:=arrAxis[AxiseNo.AxisName.AnCarryingUpDown]  , 
	axisMaster:=arrAxis[AxiseNo.VirAxisName.VirMain]  , 
	bCreatTableDone=> , 
	bCreatTableError=> , 
	bError=> );
	
fbAnCrectCamCarryingUpDown1.bCreatTableDone;
fbAnCrectCamCarryingUpDown1.bCreatTableError;
fbAnCrectCamCarryingUpDown1.bError;


//正极送纠偏搬运升降避让凸轮创建    (**********20240528SJ***************)
fbAnCrectCamCarryingUpDown3(  //避让
	bCreatTable:=fbAnCrectCamCarryingUpDown3.bCreatTable, 
	Reset:=stSysState.bReset  , 
	iTable:=TableNo.M_AnCarryingUpDown3 , 
	//fMoveLength:=arrAxisPar[AxiseNo.AxisName.AnCarryingUpDown].arrTargetPoint[10]  , //放片高度
	fSaveLength:=  arrAxisPar[AxiseNo.AxisName.AnCarryingUpDown].arrTargetPoint[10]-arrAxisPar[AxiseNo.AxisName.AnCarryingUpDown].arrTargetPoint[11] , //安全抬升高度
	//fInitLength:=arrAxisPar[AxiseNo.AxisName.AnCarryingUpDown].arrTargetPoint[4] ,//升降轴耦合初始位
	fMasterKeyPos1:=130 , //
	fMasterKeyPos2:=260 , //
	//fMasterKeyPos3:=260 , //
	//fMasterKeyPos4:=320 , //
	//fMasterKeyPos5:=359 , //
	//fMasterKeyPos6:=250 , //
	//fSlaveVelo:=0.25 , //
	axisSlave:=arrAxis[AxiseNo.AxisName.AnCarryingUpDown]  , 
	axisMaster:=arrAxis[AxiseNo.VirAxisName.VirMain]  , 
	bCreatTableDone=> , 
	bCreatTableError=> , 
	bError=> );	
fbAnCrectCamCarryingUpDown3.bCreatTableDone;
fbAnCrectCamCarryingUpDown3.bCreatTableError;
fbAnCrectCamCarryingUpDown3.bError;



//正极送纠偏搬运旋转凸轮创建 20240509 CF
fbAnCrectCamCarryingWhirling.fMoveLength:=ABS(arrAxisPar[AxiseNo.AxisName.AnCarryingWhirling].arrTargetPoint[1]-arrAxisPar[AxiseNo.AxisName.AnCarryingWhirling].arrTargetPoint[2]);
fbAnCrectCamCarryingWhirling(
	bCreatTable:=                fbAnCrectCamCarryingWhirling.bCreatTable , 
	Reset:=                          stSysState.bReset  ,  
	iTable:=                       TableNo.M_AnCarryingWhirling  , 
	fMoveLength:=             , 
	fMasterKeyPos:=          240 , //180
	
	axisMaster:=                 arrAxis[AxiseNo.VirAxisName.VirMain] ,  
    axisSlave:=                    arrAxis[AxiseNo.AxisName.AnCarryingWhirling] ,  
	bCreatTableDone=> , 
	bCreatTableError=> , 
	bError=> );

fbAnCrectCamCarryingWhirling.bCreatTableDone;
fbAnCrectCamCarryingWhirling.bCreatTableError;
fbAnCrectCamCarryingWhirling.bError;



//正极叠片搬运平移凸轮创建
fbAnCrectCamDTCarryingLine.fMoveLength:=ABS(arrAxisPar[AxiseNo.AxisName.AnDTCarryingLine].arrTargetPoint[1]-arrAxisPar[AxiseNo.AxisName.AnDTCarryingLine].arrTargetPoint[2]);
fbAnCrectCamDTCarryingLine(
	bCreatTable:=                fbAnCrectCamDTCarryingLine.bCreatTable , 
	Reset:=                          stSysState.bReset  ,  
	iTable:=                       TableNo.M_AnDTCarryingLine  , 
	fMoveLength:=             , 
	fMasterKeyPos:=          250 , //180
	
	axisMaster:=                 arrAxis[AxiseNo.VirAxisName.VirMain] ,  
    axisSlave:=                    arrAxis[AxiseNo.AxisName.AnDTCarryingLine] ,  
	bCreatTableDone=> , 
	bCreatTableError=> , 
	bError=> );
fbAnCrectCamDTCarryingLine.bCreatTableDone;
fbAnCrectCamDTCarryingLine.bCreatTableError;
fbAnCrectCamDTCarryingLine.bError;



(**********20240528SJ***************)
arrAxisPar[AxiseNo.AxisName.AnDTCarryingUpDown].arrTargetPoint[10]:=6; //等待高度  参数可调
arrAxisPar[AxiseNo.AxisName.AnDTCarryingUpDown].arrTargetPoint[11]:=18; //抬升高度  参数可调
arrAxisPar[AxiseNo.AxisName.AnDTCarryingUpDown].arrTargetPoint[4]:=arrAxisPar[AxiseNo.AxisName.AnDTCarryingUpDown].arrTargetPoint[3]-arrAxisPar[AxiseNo.AxisName.AnDTCarryingUpDown].arrTargetPoint[10];  //等待位置    以放片位为基准
//arrAxisPar[AxiseNo.AxisName.AnDTCarryingUpDown].arrTargetPoint[1]:=arrAxisPar[AxiseNo.AxisName.AnDTCarryingUpDown].arrTargetPoint[3]-arrAxisPar[AxiseNo.AxisName.AnDTCarryingUpDown].arrTargetPoint[11];  //安全位置

//正极叠片搬运升降取片凸轮创建
fbAnCrectCamDTCarryingUpDown(//取片
	bCreatTable:=fbAnCrectCamDTCarryingUpDown.bCreatTable, 
	Reset:=stSysState.bReset  , 
	iTable:=TableNo.M_AnDTCarryingUpDown , 
	fMoveLength:=arrAxisPar[AxiseNo.AxisName.AnDTCarryingUpDown].arrTargetPoint[10]-(arrAxisPar[AxiseNo.AxisName.AnDTCarryingUpDown].arrTargetPoint[3]-arrAxisPar[AxiseNo.AxisName.AnDTCarryingUpDown].arrTargetPoint[2]) , //取片高度
	fSaveLength:=arrAxisPar[AxiseNo.AxisName.AnDTCarryingUpDown].arrTargetPoint[10]-arrAxisPar[AxiseNo.AxisName.AnDTCarryingUpDown].arrTargetPoint[11]        , //安全高度
	//fInitLength:=arrAxisPar[AxiseNo.AxisName.AnDTCarryingUpDown].arrTargetPoint[4],//升降轴耦合初始位
	fMasterKeyPos1:=125 , //
	fMasterKeyPos2:=250 , //
	fMasterKeyPos3:=260 , //
	fMasterKeyPos4:= 320, //
	fMasterKeyPos5:=359 , //
	fMasterKeyPos6:= , //
	fSlaveVelo:=0.25 , //
	axisSlave:=arrAxis[AxiseNo.AxisName.AnDTCarryingUpDown]  , 
	axisMaster:=arrAxis[AxiseNo.VirAxisName.VirMain]  , 
	bCreatTableDone=> , 
	bCreatTableError=> , 
	bError=> );
fbAnCrectCamDTCarryingUpDown.bCreatTableDone;
fbAnCrectCamDTCarryingUpDown.bCreatTableError;
fbAnCrectCamDTCarryingUpDown.bError;


//正极叠片搬运升降放片凸轮创建
fbAnCrectCamDTCarryingUpDown1(//放片
	bCreatTable:=fbAnCrectCamDTCarryingUpDown1.bCreatTable, 
	Reset:=stSysState.bReset  , 
	iTable:=TableNo.M_AnDTCarryingUpDown1 , 
	fMoveLength:=arrAxisPar[AxiseNo.AxisName.AnDTCarryingUpDown].arrTargetPoint[10] ,//放片高度 
	fSaveLength:=arrAxisPar[AxiseNo.AxisName.AnDTCarryingUpDown].arrTargetPoint[10]-arrAxisPar[AxiseNo.AxisName.AnDTCarryingUpDown].arrTargetPoint[11]  , //安全高度
	//fInitLength:=arrAxisPar[AxiseNo.AxisName.AnDTCarryingUpDown].arrTargetPoint[4],//升降轴耦合初始位
	fMasterKeyPos1:=120 , //208
	fMasterKeyPos2:=250 , //256
	fMasterKeyPos3:=260 , //256
	fMasterKeyPos4:=342 , //328
	fMasterKeyPos5:=359 , //328
	fSlaveVelo:=0.25 , //
	axisSlave:=arrAxis[AxiseNo.AxisName.AnDTCarryingUpDown]  , 
	axisMaster:=arrAxis[AxiseNo.VirAxisName.VirMain]  , 
	bCreatTableDone=> , 
	bCreatTableError=> , 
	bError=> );
	
fbAnCrectCamDTCarryingUpDown1.bCreatTableDone;
fbAnCrectCamDTCarryingUpDown1.bCreatTableError;
fbAnCrectCamDTCarryingUpDown1.bError;

//正极叠片搬运升降避让凸轮创建
fbAnCrectCamDTCarryingUpDown3(//放片
	bCreatTable:=fbAnCrectCamDTCarryingUpDown3.bCreatTable, 
	Reset:=stSysState.bReset  , 
	iTable:=TableNo.M_AnDTCarryingUpDown3 , 
	//fMoveLength:=arrAxisPar[AxiseNo.AxisName.AnDTCarryingUpDown].arrTargetPoint[10] ,//放片高度 
	fSaveLength:=arrAxisPar[AxiseNo.AxisName.AnDTCarryingUpDown].arrTargetPoint[10]-arrAxisPar[AxiseNo.AxisName.AnDTCarryingUpDown].arrTargetPoint[11]  , //安全高度
	//fInitLength:=arrAxisPar[AxiseNo.AxisName.AnDTCarryingUpDown].arrTargetPoint[4],//升降轴耦合初始位
	fMasterKeyPos1:=130 , //208
	fMasterKeyPos2:=260 , //256
	//fMasterKeyPos3:=260 , //256
	//fMasterKeyPos4:=342 , //328
//	fMasterKeyPos5:=359 , //328
//	fSlaveVelo:=0.25 , //
	axisSlave:=arrAxis[AxiseNo.AxisName.AnDTCarryingUpDown]  , 
	axisMaster:=arrAxis[AxiseNo.VirAxisName.VirMain]  , 
	bCreatTableDone=> , 
	bCreatTableError=> , 
	bError=> );
	
fbAnCrectCamDTCarryingUpDown3.bCreatTableDone;
fbAnCrectCamDTCarryingUpDown3.bCreatTableError;
fbAnCrectCamDTCarryingUpDown3.bError;









An_CamTON(IN:= , PT:=T#0.5S , Q=> , ET=> );
IF Mach_Control.U.DT_iMode=3 OR Mach_Control.U.DT_iMode=0 THEN//在手动状态下
				//在触摸屏上创建正极取片凸轮
				//rAnCreate_TRIG(CLK:=Mach_Control.An_b.CreateCamStart , Q=> );
								rAnCreate_TRIG(CLK:=(Mach_Control.An_b.CreateCamStart 
									AND	NOT arrAxisCtrl[AxiseNo.AxisName.AnCarryingLine].Status.Coupled
									AND	NOT arrAxisCtrl[AxiseNo.AxisName.AnCarryingUpDown].Status.Coupled
									AND	NOT arrAxisCtrl[AxiseNo.AxisName.AnDTCarryingLine].Status.Coupled
									AND	NOT arrAxisCtrl[AxiseNo.AxisName.AnDTCarryingUpDown].Status.Coupled) , Q=> );
				IF rAnCreate_TRIG.Q THEN
					An_CamTON.IN:=FALSE;
					AnCrectCamStep0:=10;
					Mach_Control.An_b.Error[0]:=FALSE;
				END_IF
END_IF				
				//正极凸轮创建自动
				CASE AnCrectCamStep0 OF
					
							10:
									IF NOT An_CamTON.Q THEN
										An_CamTON.IN:=TRUE;
									   fbAnCrectCamCarryingLine.bCreatTable:=FALSE;//正极送片搬运平移凸轮创建
									   fbAnCrectCamCarryingUpDown.bCreatTable:=FALSE;//正极送片搬运升降取片凸轮创建
									  fbAnCrectCamUpDown_4.bCreatTable:=FALSE;//正极送片搬运升降取片凸轮创建
									  fbAnCrectCamCarryingUpDown1.bCreatTable:=FALSE;//正极送片搬运升降放片凸轮创建
									  fbAnCrectCamCarryingUpDown3.bCreatTable:=FALSE;//正极送片搬运升降放片凸轮创建								  
									  fbAnCrectCamCarryingWhirling.bCreatTable:=FALSE;//正极送片搬运旋转凸轮创建
									   fbAnCrectCamDTCarryingLine.bCreatTable :=FALSE;//正极叠片搬运平移凸轮创建
									   fbAnCrectCamDTCarryingUpDown.bCreatTable:=FALSE;//正极叠片搬运升降取片凸轮创建
									   fbAnCrectCamDTCarryingUpDown1.bCreatTable:=FALSE;//正极叠片搬运升降放片凸轮创建
									   fbAnCrectCamDTCarryingUpDown3.bCreatTable:=FALSE;//正极叠片搬运升降放片凸轮创建
									   Mach_Control.An_b.CreateCamDone:=FALSE;
									ELSE
										An_CamTON.IN:=FALSE;
									   AnCrectCamStep0:=11;
									 END_IF
							
							11:
								IF  NOT An_Cam_ton[1].Q THEN
									arrAxisCtrl[AxiseNo.AxisName.AnCarryingLine].Cmd.bStop:=TRUE;
									arrAxisCtrl[AxiseNo.AxisName.AnCarryingUpDown].Cmd.bStop:=TRUE;
									arrAxisCtrl[AxiseNo.AxisName.AnDTCarryingLine].Cmd.bStop:=TRUE;
									arrAxisCtrl[AxiseNo.AxisName.AnDTCarryingUpDown].Cmd.bStop:=TRUE;
									arrAxisCtrl[AxiseNo.AxisName.AnCarryingWhirling].Cmd.bStop:=TRUE;
									An_Cam_ton[1].IN:=TRUE;
								ELSE
									An_Cam_ton[1].IN:=FALSE;
									AnCrectCamStep0:=12;
									arrAxisCtrl[AxiseNo.AxisName.AnCarryingLine].Cmd.bStop:=FALSE;
									arrAxisCtrl[AxiseNo.AxisName.AnCarryingUpDown].Cmd.bStop:=FALSE;
									arrAxisCtrl[AxiseNo.AxisName.AnDTCarryingLine].Cmd.bStop:=FALSE;
									arrAxisCtrl[AxiseNo.AxisName.AnDTCarryingUpDown].Cmd.bStop:=FALSE;
									arrAxisCtrl[AxiseNo.AxisName.AnCarryingWhirling].Cmd.bStop:=FALSE;
								END_IF

							12:
								IF  NOT An_Cam_ton[2].Q THEN
									arrAxisCtrl[AxiseNo.AxisName.AnCarryingLine].Cmd.bReset:=TRUE;	
									arrAxisCtrl[AxiseNo.AxisName.AnCarryingUpDown].Cmd.bReset:=TRUE;
									arrAxisCtrl[AxiseNo.AxisName.AnDTCarryingLine].Cmd.bReset:=TRUE;
									arrAxisCtrl[AxiseNo.AxisName.AnDTCarryingUpDown].Cmd.bReset:=TRUE;
									arrAxisCtrl[AxiseNo.AxisName.AnCarryingWhirling].Cmd.bReset:=TRUE;
									An_Cam_ton[2].IN:=TRUE;
								 ELSE
									 An_Cam_ton[2].IN:=FALSE;
									 AnCrectCamStep0:=13;
									arrAxisCtrl[AxiseNo.AxisName.AnCarryingLine].Cmd.bReset:=FALSE;	
									arrAxisCtrl[AxiseNo.AxisName.AnCarryingUpDown].Cmd.bReset:=FALSE;
									arrAxisCtrl[AxiseNo.AxisName.AnDTCarryingLine].Cmd.bReset:=FALSE;
									arrAxisCtrl[AxiseNo.AxisName.AnDTCarryingUpDown].Cmd.bReset:=FALSE;
									arrAxisCtrl[AxiseNo.AxisName.AnCarryingWhirling].Cmd.bReset:=FALSE;
								 END_IF
								 
							13:
									arrAxisCtrl[AxiseNo.AxisName.AnCarryingLine].Cmd.bEnable:=TRUE;
									arrAxisCtrl[AxiseNo.AxisName.AnCarryingUpDown].Cmd.bEnable:=TRUE;
									arrAxisCtrl[AxiseNo.AxisName.AnDTCarryingLine].Cmd.bEnable:=TRUE;
									arrAxisCtrl[AxiseNo.AxisName.AnDTCarryingUpDown].Cmd.bEnable:=TRUE;
									arrAxisCtrl[AxiseNo.AxisName.AnCarryingWhirling].Cmd.bEnable:=TRUE;
									IF arrAxisCtrl[AxiseNo.AxisName.AnCarryingLine].Status.Enabled AND arrAxisCtrl[AxiseNo.AxisName.AnCarryingUpDown].Status.Enabled AND
										arrAxisCtrl[AxiseNo.AxisName.AnDTCarryingLine].Status.Enabled AND arrAxisCtrl[AxiseNo.AxisName.AnDTCarryingUpDown].Status.Enabled
										AND arrAxisCtrl[AxiseNo.AxisName.AnCarryingWhirling].Status.Enabled THEN
										 AnCrectCamStep0:=20;
									END_IF


		   
							20://创建凸轮
									  fbAnCrectCamCarryingLine.bCreatTable:=TRUE;//正极送片搬运平移凸轮创建
									  fbAnCrectCamCarryingUpDown.bCreatTable:=TRUE;//正极送片搬运升降取片凸轮创建
									  fbAnCrectCamUpDown_4.bCreatTable:=TRUE;//正极送片搬运升降取片凸轮创建
									  
									  fbAnCrectCamCarryingUpDown1.bCreatTable:=TRUE;//正极送片搬运升降放片凸轮创建
									   fbAnCrectCamCarryingUpDown3.bCreatTable:=TRUE;//正极送片搬运升降放片凸轮创建
									  fbAnCrectCamCarryingWhirling.bCreatTable:=TRUE;//正极送片搬运旋转凸轮创建
									   fbAnCrectCamDTCarryingLine.bCreatTable :=TRUE;//正极叠片搬运平移凸轮创建
									   fbAnCrectCamDTCarryingUpDown.bCreatTable:=TRUE;//正极叠片搬运升降取片凸轮创建
									   fbAnCrectCamDTCarryingUpDown1.bCreatTable:=TRUE;//正极叠片搬运升降放片凸轮创建
									    fbAnCrectCamDTCarryingUpDown3.bCreatTable:=TRUE;//正极叠片搬运升降放片凸轮创建
									   
									   Mach_Control.An_b.CreateCamDone:=FALSE;
									   AnCrectCamStep0:=30;
							30://等待凸轮创建完成
									IF fbAnCrectCamCarryingLine.bCreatTableDone AND fbAnCrectCamUpDown_4.bCreatTableDone(*fbAnCrectCamCarryingUpDown.bCreatTableDone*) AND fbAnCrectCamCarryingUpDown1.bCreatTableDone  AND fbAnCrectCamCarryingWhirling.bCreatTableDone AND 
										fbAnCrectCamDTCarryingLine.bCreatTableDone AND fbAnCrectCamDTCarryingUpDown.bCreatTableDone AND fbAnCrectCamDTCarryingUpDown1.bCreatTableDone  AND 
                                        fbAnCrectCamCarryingUpDown3.bCreatTableDone AND  fbAnCrectCamDTCarryingUpDown3.bCreatTableDone  THEN
										Mach_Control.An_b.CreateCamDone:=TRUE;
										 AnCrectCamStep0:=6666;
										ELSE
												IF fbAnCrectCamCarryingLine.bCreatTableError OR fbAnCrectCamCarryingUpDown.bCreatTableError OR fbAnCrectCamCarryingUpDown1.bCreatTableError OR fbAnCrectCamCarryingWhirling.bCreatTableError OR 
													fbAnCrectCamCarryingLine.bCreatTableError OR fbAnCrectCamDTCarryingUpDown.bCreatTableError OR fbAnCrectCamDTCarryingUpDown1.bCreatTableError OR fbAnCrectCamUpDown_4.bCreatTableError OR 
                                                  fbAnCrectCamCarryingUpDown3.bCreatTableError OR  fbAnCrectCamDTCarryingUpDown3.bCreatTableError   THEN
													Mach_Control.An_b.Error[0]:=TRUE;//正极取片凸轮创建失败报警
													AnCrectCamStep0:=9999;
												END_IF
									END_IF
				END_CASE







(***********************************正极凸轮耦合***********************************************)
(*
      fbAnCamInCarryingLine                      :FB_CamIn ;    
      fbAnCamInCarryingUpDown               :FB_CamIn ;    
      fbAnCamInDTCarryingLine                    :FB_CamIn ;    
      fbAnCamInDTCarryingUpDown             :FB_CamIn ;     
*)
//正极送片搬运平移凸轮耦合
fbAnCamInCarryingLine.ParCamIn.SlaveScaling;
fbAnCamInCarryingLine.ParCamIn.MasterScaling:=fAnScaling;//20240508 CF
fbAnCamInCarryingLine(
	Reset:=                      stSysState.bReset  , 
	bCamInExecute:=       fbAnCamInCarryingLine.bCamInExecute, 
	iTable1:=                   TableNo.M_AnCarryingLine  , 
	iTable2:=                   , 
	iTableSel:=                 , 
	ParCamIn:= , 
  	axisMaster:=            arrAxis[AxiseNo.VirAxisName.VirMain] ,  
	axisSlave:=               arrAxis[AxiseNo.AxisName.AnCarryingLine] ,  
	bError=> , 
	bReady=> , 
	bInSync=> );

(*Mach_Control.An_b.Error[9]:=*)fbAnCamInCarryingLine.bError;
fbAnCamInCarryingLine.bReady;
fbAnCamInCarryingLine.bInSync;

//正极送片搬运升降凸轮耦合
fbAnCamInCarryingUpDown(
	Reset:=                      stSysState.bReset  , 
	bCamInExecute:=       fbAnCamInCarryingUpDown.bCamInExecute, 
	iTable1:=                   TableNo.M_AnCarryingUpDown  , 
	iTable2:=                    TableNo.M_AnCarryingUpDown1 , 
	iTable3:=                    TableNo.M_AnCarryingUpDown3 , 
	iTableSel:=                  , 
	ParCamIn:=                  , 
  	axisMaster:=            arrAxis[AxiseNo.VirAxisName.VirMain] ,  
	axisSlave:=               arrAxis[AxiseNo.AxisName.AnCarryingUpDown] ,  
	bError=> , 
	bReady=> , 
	bInSync=> );

(*Mach_Control.An_b.Error[10]:=*)fbAnCamInCarryingUpDown.bError;
fbAnCamInCarryingUpDown.bReady;
fbAnCamInCarryingUpDown.bInSync;
//正极送片搬运旋转凸轮耦合
fbAnCamInCarryingWhirling.ParCamIn.SlaveScaling;
fbAnCamInCarryingWhirling.ParCamIn.MasterScaling:=fAnScaling;//20240508 CF
fbAnCamInCarryingWhirling(
	Reset:=                      stSysState.bReset  , 
	bCamInExecute:=       fbAnCamInCarryingWhirling.bCamInExecute, 
	iTable1:=                   TableNo.M_AnCarryingWhirling  , 
	iTable2:=                    , 
	iTableSel:=                  , 
	ParCamIn:=                  , 
  	axisMaster:=            arrAxis[AxiseNo.VirAxisName.VirMain] ,  
	axisSlave:=               arrAxis[AxiseNo.AxisName.AnCarryingWhirling] ,  
	bError=> , 
	bReady=> , 
	bInSync=> );

(*Mach_Control.An_b.Error[11]:=*)fbAnCamInCarryingWhirling.bError;
fbAnCamInCarryingWhirling.bReady;
fbAnCamInCarryingWhirling.bInSync;



//正极叠片搬运平移凸轮耦合
fbAnCamInDTCarryingLine.ParCamIn.SlaveScaling;
fbAnCamInDTCarryingLine(
	Reset:=                      stSysState.bReset  , 
	bCamInExecute:=       fbAnCamInDTCarryingLine.bCamInExecute, 
	iTable1:=                   TableNo.M_AnDTCarryingLine  , 
	iTable2:=                   , 
	iTableSel:=                 , 
	ParCamIn:=                , 
  	axisMaster:=            arrAxis[AxiseNo.VirAxisName.VirMain] ,  
	axisSlave:=               arrAxis[AxiseNo.AxisName.AnDTCarryingLine] ,  
	bError=> , 
	bReady=> , 
	bInSync=> );
(*Mach_Control.An_b.Error[12]:=*)fbAnCamInDTCarryingLine.bError;
fbAnCamInDTCarryingLine.bReady;
fbAnCamInDTCarryingLine.bInSync;


//正极叠片搬运升降凸轮耦合
fbAnCamInDTCarryingUpDown(
	Reset:=                      stSysState.bReset  , 
	bCamInExecute:=       fbAnCamInDTCarryingUpDown.bCamInExecute, 
	iTable1:=                   TableNo.M_AnDTCarryingUpDown  , 
	iTable2:=                    TableNo.M_AnDTCarryingUpDown1, 
	iTable3:=                    TableNo.M_AnDTCarryingUpDown3, 
	iTableSel:=                  , 
	ParCamIn:=                  , 
  	axisMaster:=            arrAxis[AxiseNo.VirAxisName.VirMain] ,  
	axisSlave:=               arrAxis[AxiseNo.AxisName.AnDTCarryingUpDown] ,  
	bError=> , 
	bReady=> , 
	bInSync=> );

(*Mach_Control.An_b.Error[13]:=*)fbAnCamInDTCarryingUpDown.bError;
fbAnCamInDTCarryingUpDown.bReady;
fbAnCamInDTCarryingUpDown.bInSync;


IF fbAnCamInCarryingLine.bError OR fbAnCamInCarryingUpDown.bError OR fbAnCamInCarryingWhirling.bError OR fbAnCamInDTCarryingLine.bError OR fbAnCamInDTCarryingUpDown.bError THEN
		Mach_Control.An_b.Error[11]:=TRUE;//正极有凸轮耦合报警
	ELSE		
		Mach_Control.An_b.Error[11]:=FALSE;
END_IF
END_ACTION

ACTION An_Conditions:
//正极纠偏平台允许放料条件
IF  NOT Mach_Control.An_b.An_deviationFalg AND arrAxisCtrl[AxiseNo.AxisName.AndeviationX1].Status.Homed AND NOT arrAxisCtrl[AxiseNo.AxisName.AndeviationX1].Status.Error AND 
	arrAxisCtrl[AxiseNo.AxisName.AndeviationX1].Status.NoMoving AND arrAxisCtrl[AxiseNo.AxisName.AndeviationX1].Cmd.arrbRealPoint[1] AND 
	arrAxisCtrl[AxiseNo.AxisName.AndeviationX2].Status.Homed AND NOT arrAxisCtrl[AxiseNo.AxisName.AndeviationX2].Status.Error AND 
	arrAxisCtrl[AxiseNo.AxisName.AndeviationX2].Status.NoMoving AND arrAxisCtrl[AxiseNo.AxisName.AndeviationX2].Cmd.arrbRealPoint[1] AND 
	arrAxisCtrl[AxiseNo.AxisName.AndeviationY].Status.Homed AND NOT arrAxisCtrl[AxiseNo.AxisName.AndeviationY].Status.Error AND 
	arrAxisCtrl[AxiseNo.AxisName.AndeviationY].Status.NoMoving AND arrAxisCtrl[AxiseNo.AxisName.AndeviationY].Cmd.arrbRealPoint[1] THEN
	Mach_Control.An_b.An_deviationFPOK:=TRUE;
ELSE
	Mach_Control.An_b.An_deviationFPOK:=FALSE;
END_IF 
(*
//正极纠偏平台允许取料条件
IF Mach_Control.An_b.An_deviationFalg AND  (Mach_Control.An_b.An_deviationDone OR Mach_Control.U.CCD_ChosesHMI OR Mach_Control.U.EmptyRunMode) THEN
	Mach_Control.An_b.An_deviationDPOK:=TRUE;
ELSE
	Mach_Control.An_b.An_deviationDPOK:=FALSE;
END_IF
*)
//正极送片搬运平移在安全位，正极送片升降在安全位，允许正极叠片搬运平移到纠偏位
IF arrAxisCtrl[AxiseNo.AxisName.AnCarryingLine].Status.Homed AND arrAxisCtrl[AxiseNo.AxisName.AnCarryingLine].Status.NoMoving AND arrAxisCtrl[AxiseNo.AxisName.AnCarryingLine].Cmd.arrbRealPoint[1] AND 
 	arrAxisCtrl[AxiseNo.AxisName.AnDTCarryingUpDown].Status.Homed AND arrAxisCtrl[AxiseNo.AxisName.AnDTCarryingUpDown].Status.NoMoving AND arrAxisCtrl[AxiseNo.AxisName.AnDTCarryingUpDown].Cmd.arrbRealPoint[1] THEN
	Mach_Control.An_b.CarryingSafepos[0]:=TRUE;
ELSE
	Mach_Control.An_b.CarryingSafepos[0]:=FALSE;
END_IF
//正极隔膜平移在负极片位、正极送片搬运升降在安全位，允许正极叠片搬动至叠台位
IF arrAxisCtrl[AxiseNo.AxisName.SEPTATLine].Status.Homed AND arrAxisCtrl[AxiseNo.AxisName.SEPTATLine].Status.NoMoving AND arrAxisCtrl[AxiseNo.AxisName.SEPTATLine].Cmd.arrbRealPoint[2] AND 
	 	arrAxisCtrl[AxiseNo.AxisName.AnDTCarryingUpDown].Status.Homed AND arrAxisCtrl[AxiseNo.AxisName.AnDTCarryingUpDown].Status.NoMoving AND arrAxisCtrl[AxiseNo.AxisName.AnDTCarryingUpDown].Cmd.arrbRealPoint[1] THEN
	Mach_Control.An_b.CarryingSafepos[1]:=TRUE;
ELSE		
	Mach_Control.An_b.CarryingSafepos[1]:=FALSE;
END_IF
//正极送片搬运升降在安全位，允许正极送片搬运平移至取流水线极片位
IF  arrAxisCtrl[AxiseNo.AxisName.AnCarryingUpDown].Status.Homed AND arrAxisCtrl[AxiseNo.AxisName.AnCarryingUpDown].Status.NoMoving AND arrAxisCtrl[AxiseNo.AxisName.AnCarryingUpDown].Cmd.arrbRealPoint[1] THEN
		Mach_Control.An_b.CarryingSafepos[2]:=TRUE;
ELSE
		Mach_Control.An_b.CarryingSafepos[2]:=FALSE;	
END_IF
//正极送片搬运升降在安全位、正极叠片搬运平移在安全位，允许正极送片搬运平移纠偏位
IF  arrAxisCtrl[AxiseNo.AxisName.AnCarryingUpDown].Status.Homed AND arrAxisCtrl[AxiseNo.AxisName.AnCarryingUpDown].Status.NoMoving AND arrAxisCtrl[AxiseNo.AxisName.AnCarryingUpDown].Cmd.arrbRealPoint[1] AND 
 	arrAxisCtrl[AxiseNo.AxisName.AnDTCarryingLine].Status.Homed AND arrAxisCtrl[AxiseNo.AxisName.AnDTCarryingLine].Status.NoMoving AND arrAxisCtrl[AxiseNo.AxisName.AnDTCarryingLine].Cmd.arrbRealPoint[2]  THEN
		Mach_Control.An_b.CarryingSafepos[3]:=TRUE;
ELSE
		Mach_Control.An_b.CarryingSafepos[3]:=FALSE;	
END_IF
//允许正极纠偏平台移动
IF arrAxisCtrl[AxiseNo.AxisName.AnCarryingUpDown].Status.Homed AND arrAxisCtrl[AxiseNo.AxisName.AnCarryingLine].Status.Homed AND 
	((arrAxisCtrl[AxiseNo.AxisName.AnCarryingUpDown].Status.fSetPos<=arrAxisPar[AxiseNo.AxisName.AnCarryingUpDown].arrTargetPoint[4]+2) OR arrAxisCtrl[AxiseNo.AxisName.AnCarryingLine].Cmd.arrbGoSetPos[1]) AND 
	((arrAxisCtrl[AxiseNo.AxisName.AnDTCarryingUpDown].Status.fSetPos<=arrAxisPar[AxiseNo.AxisName.AnDTCarryingUpDown].arrTargetPoint[4]+2) OR arrAxisCtrl[AxiseNo.AxisName.AnDTCarryingLine].Cmd.arrbGoSetPos[2])THEN
	Mach_Control.An_b.CarryingSafepos[4]:=TRUE;
ELSE
	Mach_Control.An_b.CarryingSafepos[4]:=FALSE;
END_IF
//正极取流水线机械手在安全位，允许模切流水线移动
(*
IF arrAxisCtrl[AxiseNo.AxisName.AnCarryingUpDown].Status.Homed AND NOT Mach_Control.An_b.An_MainBelting AND
	(arrAxisCtrl[AxiseNo.AxisName.AnCarryingUpDown].Status.fSetPos<=arrAxisPar[AxiseNo.AxisName.AnCarryingUpDown].arrTargetPoint[4]+0.2 OR arrAxisCtrl[AxiseNo.AxisName.AnCarryingLine].Cmd.arrbRealPoint[2]) THEN
	Mach_Control.An_b.AN_BeltSafe:=TRUE;
ELSE
	Mach_Control.An_b.AN_BeltSafe:=FALSE;
END_IF
*)
(*
IF  Mach_Control.An_b.An_MainBelting  THEN
	Mach_Control.An_b.AN_BeltSafe:=TRUE;
ELSIF NOT Mach_Control.An_b.An_MainBelting AND  arrAxisCtrl[AxiseNo.AxisName.AnCarryingUpDown].Cmd.arrbRealPoint[4] THEN
	Mach_Control.An_b.AN_BeltSafe:=FALSE;
END_IF
*)
IF  Mach_Control.An_b.An_MainBelting  THEN
	Mach_Control.An_b.AN_BeltSafe:=TRUE;
ELSE
	Mach_Control.An_b.AN_BeltSafe:=FALSE;
END_IF

//正极主流水线取片完成延时复位
An_BeltTon(IN:=Mach_Control.An_b.AN_BeltDone , PT:=T#0.1S , Q=> , ET=> );
IF An_BeltTon.Q THEN
	Mach_Control.An_b.AN_BeltDone :=FALSE;
END_IF


//正极跳取条件1:空跑(空叠隔膜)
An_JumpRules[1]:=Mach_Control.U.EmptyRunMode OR (Mach_Control.DT_b.SinStepMode AND An_Step0<>150);
//正极跳取条件2:手动
An_JumpRules[2]:=Mach_Control.U.DT_iMode<>1;
//正极跳取条件3:叠完电芯后空叠隔膜
An_JumpRules[3]:=Mach_Control.DT_b.DP_Mode AND Mach_Control.An_b.An_Quantited=Par.stDT_date.An_Quantity AND Par.stDT_date.An_Quantity<>0  ;
//正极跳取条件4:叠完电芯后下料
An_JumpRules[4]:=DP_Step0>=6000;//(DP_Step0>=6030 AND DP_Step0<6041) ;
//正极跳取条件5:正极剔废,
An_JumpRules[5]:=(An_Step2<>0 AND An_Step2<>6666) ; 
//正极跳取条件6:接带、蓝胶判断
An_JumpRules[6]:=Bnt_Blueflaging AND Mach_Control.Ca_b.Ca_Quantited>=Par.stDT_date.DT_Overhang_SUM AND Par.stDT_date.DT_Overhang_SUM>0 
				AND Mach_Control.Ca_b.Ca_Quantited>Mach_Control.An_b.An_Quantited AND An_StandbyStep1<1000;//已经进入取片流程则取完当前片
//正极跳取条件7:取片升降有片
An_JumpRules[7]:= Mach_Control.An_b.An_CarryingFalg  ;
//正极跳取条件8:对齐度踢废
An_JumpRules[8]:=Mach_Control.DT_b.DT_Oerhang_Z=2 AND  Par.stDT_date.DT_Overhang_SUM>0 AND Mach_Control.Ca_b.Ca_Quantited>=Par.stDT_date.DT_Overhang_SUM
				AND Mach_Control.An_b.An_Quantited<Mach_Control.Ca_b.Ca_Quantited  AND  Mach_Control.DT_b.DT_CellNG_TF AND Mach_Control.DT_b.Overhang_TF 
				AND((NOT Mach_Control.DT_b.FirstEmpFold AND   bFirstFoldFinish[1]) OR (Mach_Control.DT_b.FirstEmpFold)) AND An_StandbyStep1<1000;//已经进入取片流程则取完当前片
//正极跳取条件9:负极剔废
An_JumpRules[9]:=(Ca_Step2<>0 AND Ca_Step2<>6666) ;
//正极跳取条件10:首层空叠隔膜流程
An_JumpRules[10]:=NOT bFirstFoldFinish[1]AND NOT Mach_Control.DT_b.FirstEmpFold ; 			
//正极跳取条件
Mach_Control.An_b.JumpPiceReady:=An_JumpRules[1] OR An_JumpRules[2] OR An_JumpRules[3] OR An_JumpRules[4] OR An_JumpRules[5]
				OR An_JumpRules[6] OR An_JumpRules[7] OR An_JumpRules[8]  OR An_JumpRules[9] OR An_JumpRules[10] OR DP_Step0=162;	//速度不一样如果平移没到位放弃取片 20240509 CF	
//正极取片条件
Mach_Control.An_b.GetPiceReady:=NOT Mach_Control.An_b.JumpPiceReady (*AND  arrAxisCtrl[AxiseNo.AxisName.AnCarryingUpDown].Cmd.arrbRealPoint[4]*)
				AND ABS(arrAxisCtrl[AxiseNo.AxisName.AnCarryingLine].Status.fSetPos-arrAxisPar[AxiseNo.AxisName.AnCarryingLine].arrTargetPoint[1])<0.5 AND  arrAxisCtrl[AxiseNo.AxisName.AnCarryingWhirling].Cmd.arrbRealPoint[1]
				AND Mach_Control.U.DT_iMode=1 AND NOT Mach_Control.An_b.An_CarryingFalg ;//20240509 CF 升降位置判断屏蔽
		
(*				
////////////////判断叠台是否需要极片
//南昌原版
JumpPiceReady_temp1:=Mach_Control.An_b.An_Quantited<Mach_Control.Ca_b.Ca_Quantited AND Par.stDT_date.An_Quantity<>0  AND
 	 				 Par.stDT_date.Ca_Quantity <>0 AND  Mach_Control.DT_b.DT_CellNG_TF AND
	 				 Mach_Control.Ca_b.Ca_Quantited>=Par.stDT_date.DT_Overhang_SUM AND Par.stDT_date.DT_Overhang_SUM>0  AND
     				 Mach_Control.DT_b.DT_Oerhang_Z=2 AND  NOT Mach_Control.U.EmptyRunMode;

JumpPiceReady_temp2:=Bnt_Blueflaging AND ((Mach_Control.An_b.An_Quantited=0 AND Mach_Control.Ca_b.Ca_Quantited=0) OR
 					 Mach_Control.Ca_b.Ca_Quantited>Mach_Control.An_b.An_Quantited);

JumpPiceReady_temp3:= Mach_Control.An_b.An_Quantited >= Par.stDT_date.An_Quantity  AND
  					  Mach_Control.Ca_b.Ca_Quantited >= Par.stDT_date.Ca_Quantity AND
                      Par.stDT_date.An_Quantity<>0  AND Par.stDT_date.Ca_Quantity <>0;
					  
JumpPiceReady_temp4:= (Ca_Step2<>0 AND Ca_Step2<>6666 AND Mach_Control.U.DT_iMode=1)OR (Mach_Control.An_b.An_Quantited >= Par.stDT_date.An_Quantity 
					 AND  Mach_Control.Ca_b.Ca_Quantited >= (Par.stDT_date.Ca_Quantity-1)) OR
					   (Bnt_Blueflaging AND Mach_Control.Ca_b.Ca_Quantited>=Par.stDT_date.DT_Overhang_SUM AND Par.stDT_date.DT_Overhang_SUM>0);

					   
//正极送片搬运搬运取片准备好
IF Mach_Control.U.DT_iMode=1 AND NOT Mach_Control.An_b.An_CarryingFalg AND NOT JumpPiceReady_temp4 AND (DP_Step0<>6030 AND DP_Step0<>6040 AND 
Mach_Control.An_b.An_Quantited <= Par.stDT_date.An_Quantity  AND  Mach_Control.Ca_b.Ca_Quantited < Par.stDT_date.Ca_Quantity) AND
   arrAxisCtrl[AxiseNo.AxisName.AnCarryingUpDown].Cmd.arrbRealPoint[4] AND arrAxisCtrl[AxiseNo.AxisName.AnCarryingUpDown].Status.Homed AND
   arrAxisCtrl[AxiseNo.AxisName.AnCarryingLine].Cmd.arrbRealPoint[1] AND arrAxisCtrl[AxiseNo.AxisName.AnCarryingLine].Status.Homed AND
   arrAxisCtrl[AxiseNo.AxisName.AnCarryingWhirling].Cmd.arrbRealPoint[1]AND arrAxisCtrl[AxiseNo.AxisName.AnCarryingWhirling].Status.Homed  THEN
   Mach_Control.An_b.GetPiceReady:=TRUE;
ELSE
   Mach_Control.An_b.GetPiceReady:=FALSE;	
END_IF

//正极送片搬运不取片
IF Mach_Control.U.DT_iMode<>1 OR Mach_Control.An_b.An_CarryingFalg OR JumpPiceReady_temp1 OR JumpPiceReady_temp2 OR JumpPiceReady_temp3 OR JumpPiceReady_temp4 OR Mach_Control.U.EmptyRunMode THEN
	Mach_Control.An_b.JumpPiceReady:=TRUE;
ELSE
	Mach_Control.An_b.JumpPiceReady:=FALSE;	
END_IF


//合肥原版
(*
(********************正极取片准备好********************)															
Mach_Control.An_b.GetPiceReady:=NOT Mach_Control.An_b.JumpPiceReady AND 
							arrAxisCtrl[AxiseNo.AxisName.AnCarryingUpDown].Cmd.arrbRealPoint[4] AND arrAxisCtrl[AxiseNo.AxisName.AnCarryingUpDown].Status.Homed AND
							arrAxisCtrl[AxiseNo.AxisName.AnCarryingLine].Cmd.arrbRealPoint[1] AND arrAxisCtrl[AxiseNo.AxisName.AnCarryingLine].Status.Homed AND
							arrAxisCtrl[AxiseNo.AxisName.AnCarryingWhirling].Cmd.arrbRealPoint[1]AND arrAxisCtrl[AxiseNo.AxisName.AnCarryingWhirling].Status.Homed AND 
							(DP_Step0<>6030 AND DP_Step0<>6040)  ;													

(********************正极放弃取片********************)
Mach_Control.An_b.JumpPiceReady:=Mach_Control.U.DT_iMode<>1 OR Mach_Control.An_b.An_CarryingFalg OR Blueflaging OR Mach_Control.U.EmptyRunMode
															OR Mach_Control.An_b.An_Quantited=Par.stDT_date.An_Quantity;
*)

*)


/////////////////////////////////////////////////////////////
/////////////////////////////////////////////////////////
////////////////////////////////////////////电机条件
//正极送片搬运平移
IF arrAxisCtrl[AxiseNo.AxisName.AnCarryingUpDown].Status.fSetPos<=arrAxisPar[AxiseNo.AxisName.AnCarryingUpDown].arrTargetPoint[4]+1 AND
 	arrAxisCtrl[AxiseNo.AxisName.AnCarryingUpDown].Status.Homed AND arrAxisCtrl[AxiseNo.AxisName.AnCarryingUpDown].Status.NoMoving	AND Mach_Control.U.DT_iMode=3 THEN
arrAxisCtrl[AxiseNo.AxisName.AnCarryingLine].Cmd.Home_Condition:=TRUE;
ELSE
arrAxisCtrl[AxiseNo.AxisName.AnCarryingLine].Cmd.Home_Condition:=FALSE;	
END_IF

IF arrAxisCtrl[AxiseNo.AxisName.AnCarryingUpDown].Status.fSetPos<=arrAxisPar[AxiseNo.AxisName.AnCarryingUpDown].arrTargetPoint[4]+1 AND
	arrAxisCtrl[AxiseNo.AxisName.AnCarryingUpDown].Status.Homed AND arrAxisCtrl[AxiseNo.AxisName.AnCarryingUpDown].Status.NoMoving AND Mach_Control.U.DT_iMode=3 
    AND 	arrCyCtrl[arrCyNo.CylinderName.AnScrapbinCy].Io.DIOnSwitch  THEN
arrAxisCtrl[AxiseNo.AxisName.AnCarryingLine].Cmd.GoPoint_Condition[1]:=TRUE;
ELSE
arrAxisCtrl[AxiseNo.AxisName.AnCarryingLine].Cmd.GoPoint_Condition[1]:=FALSE;	
END_IF

IF arrAxisCtrl[AxiseNo.AxisName.AnCarryingUpDown].Status.fSetPos<=arrAxisPar[AxiseNo.AxisName.AnCarryingUpDown].arrTargetPoint[4]+1 AND arrAxisCtrl[AxiseNo.AxisName.AnCarryingUpDown].Status.Homed  AND
	 arrAxisCtrl[AxiseNo.AxisName.AnCarryingLine].Status.Homed AND Mach_Control.U.DT_iMode=3 AND 	arrCyCtrl[arrCyNo.CylinderName.AnScrapbinCy].Io.DIOnSwitch AND
	 arrAxisCtrl[AxiseNo.AxisName.AnDTCarryingLine].Status.Homed AND arrAxisCtrl[AxiseNo.AxisName.AnDTCarryingLine].Cmd.arrbRealPoint[2] THEN//比较值要根据实际值修改
	arrAxisCtrl[AxiseNo.AxisName.AnCarryingLine].Cmd.GoPoint_Condition[2]:=TRUE;
ELSE
	arrAxisCtrl[AxiseNo.AxisName.AnCarryingLine].Cmd.GoPoint_Condition[2]:=FALSE;	
END_IF

//正极送片搬运升降
IF Mach_Control.U.DT_iMode=3  THEN
	arrAxisCtrl[AxiseNo.AxisName.AnCarryingUpDown].Cmd.Home_Condition:=TRUE;
ELSE
	arrAxisCtrl[AxiseNo.AxisName.AnCarryingUpDown].Cmd.Home_Condition:=FALSE;	
END_IF

IF Mach_Control.U.DT_iMode=3 AND arrAxisCtrl[AxiseNo.AxisName.AnCarryingUpDown].Status.Homed THEN
	arrAxisCtrl[AxiseNo.AxisName.AnCarryingUpDown].Cmd.GoPoint_Condition[1]:=TRUE;
ELSE
	arrAxisCtrl[AxiseNo.AxisName.AnCarryingUpDown].Cmd.GoPoint_Condition[1]:=FALSE;	
END_IF

IF (*arrAxisCtrl[AxiseNo.AxisName.AnCarryingLine].Cmd.arrbRealPoint[1] AND*)  Mach_Control.U.DT_iMode=3 AND arrAxisCtrl[AxiseNo.AxisName.AnCarryingUpDown].Status.Homed THEN
	arrAxisCtrl[AxiseNo.AxisName.AnCarryingUpDown].Cmd.GoPoint_Condition[2]:=TRUE;
ELSE
	arrAxisCtrl[AxiseNo.AxisName.AnCarryingUpDown].Cmd.GoPoint_Condition[2]:=FALSE;	
END_IF

IF (*arrAxisCtrl[AxiseNo.AxisName.AnCarryingLine].Cmd.arrbRealPoint[2] AND*)  Mach_Control.U.DT_iMode=3 AND arrAxisCtrl[AxiseNo.AxisName.AnCarryingUpDown].Status.Homed THEN
	arrAxisCtrl[AxiseNo.AxisName.AnCarryingUpDown].Cmd.GoPoint_Condition[3]:=TRUE;
ELSE
	arrAxisCtrl[AxiseNo.AxisName.AnCarryingUpDown].Cmd.GoPoint_Condition[3]:=FALSE;	
END_IF

IF (*arrAxisCtrl[AxiseNo.AxisName.AnCarryingLine].Cmd.arrbRealPoint[1] AND*)  Mach_Control.U.DT_iMode=3 AND arrAxisCtrl[AxiseNo.AxisName.AnCarryingUpDown].Status.Homed THEN
	arrAxisCtrl[AxiseNo.AxisName.AnCarryingUpDown].Cmd.GoPoint_Condition[4]:=TRUE;
ELSE
	arrAxisCtrl[AxiseNo.AxisName.AnCarryingUpDown].Cmd.GoPoint_Condition[4]:=FALSE;	
END_IF

//正极送片搬运旋转
IF Mach_Control.U.DT_iMode=3 AND
 	arrAxisCtrl[AxiseNo.AxisName.AnCarryingUpDown].Status.fSetPos <= arrAxisPar[AxiseNo.AxisName.AnCarryingUpDown].arrTargetPoint[1]+1 AND 
	arrAxisCtrl[AxiseNo.AxisName.AnCarryingUpDown].Status.Homed AND arrCyCtrl[arrCyNo.CylinderName.AnScrapbinCy].Io.DIOnSwitch   THEN
	arrAxisCtrl[AxiseNo.AxisName.AnCarryingWhirling].Cmd.Home_Condition:=TRUE;
ELSE
	arrAxisCtrl[AxiseNo.AxisName.AnCarryingWhirling].Cmd.Home_Condition:=FALSE;	
END_IF


IF Mach_Control.U.DT_iMode=3 AND
 	arrAxisCtrl[AxiseNo.AxisName.AnCarryingUpDown].Status.fSetPos <= arrAxisPar[AxiseNo.AxisName.AnCarryingUpDown].arrTargetPoint[1]+1 AND 
	arrAxisCtrl[AxiseNo.AxisName.AnCarryingUpDown].Status.Homed AND arrCyCtrl[arrCyNo.CylinderName.AnScrapbinCy].Io.DIOnSwitch    THEN
	   arrAxisCtrl[AxiseNo.AxisName.AnCarryingWhirling].Cmd.JogP_Condition:=TRUE;
	   arrAxisCtrl[AxiseNo.AxisName.AnCarryingWhirling].Cmd.JogN_Condition:=TRUE;
 ELSE 
	   arrAxisCtrl[AxiseNo.AxisName.AnCarryingWhirling].Cmd.JogP_Condition:=FALSE;
	   arrAxisCtrl[AxiseNo.AxisName.AnCarryingWhirling].Cmd.JogN_Condition:=FALSE;
 END_IF

IF Mach_Control.U.DT_iMode=3 AND 
	(arrAxisCtrl[AxiseNo.AxisName.AnCarryingUpDown].Cmd.arrbRealPoint[1] (*OR arrAxisCtrl[AxiseNo.AxisName.AnCarryingUpDown].Cmd.arrbRealPoint[4]*))AND
	arrAxisCtrl[AxiseNo.AxisName.AnCarryingUpDown].Status.Homed AND arrAxisCtrl[AxiseNo.AxisName.AnCarryingWhirling].Status.Homed AND 
    arrCyCtrl[arrCyNo.CylinderName.AnScrapbinCy].Io.DIOnSwitch   THEN
	arrAxisCtrl[AxiseNo.AxisName.AnCarryingWhirling].Cmd.GoPoint_Condition[1]:=TRUE;
ELSE
	arrAxisCtrl[AxiseNo.AxisName.AnCarryingWhirling].Cmd.GoPoint_Condition[1]:=FALSE;	
END_IF

IF Mach_Control.U.DT_iMode=3 AND 
	(arrAxisCtrl[AxiseNo.AxisName.AnCarryingUpDown].Cmd.arrbRealPoint[1] (*OR arrAxisCtrl[AxiseNo.AxisName.AnCarryingUpDown].Cmd.arrbRealPoint[4]*)) AND
	arrAxisCtrl[AxiseNo.AxisName.AnCarryingUpDown].Status.Homed AND arrAxisCtrl[AxiseNo.AxisName.AnCarryingWhirling].Status.Homed AND
   arrCyCtrl[arrCyNo.CylinderName.AnScrapbinCy].Io.DIOnSwitch  THEN
	arrAxisCtrl[AxiseNo.AxisName.AnCarryingWhirling].Cmd.GoPoint_Condition[2]:=TRUE;
ELSE
	arrAxisCtrl[AxiseNo.AxisName.AnCarryingWhirling].Cmd.GoPoint_Condition[2]:=FALSE;	
END_IF

//正极纠偏平台X1
IF Mach_Control.U.DT_iMode=3  OR  (DP_Step0>=6015 AND   DP_Step0<=6041)   THEN
	arrAxisCtrl[AxiseNo.AxisName.AndeviationX1].Cmd.Home_Condition:=TRUE;
ELSE
	arrAxisCtrl[AxiseNo.AxisName.AndeviationX1].Cmd.Home_Condition:=FALSE;	
END_IF

IF Mach_Control.U.DT_iMode=3 AND arrAxisCtrl[AxiseNo.AxisName.AndeviationX1].Status.Homed THEN
	arrAxisCtrl[AxiseNo.AxisName.AndeviationX1].Cmd.GoPoint_Condition[1]:=TRUE;
ELSE
	arrAxisCtrl[AxiseNo.AxisName.AndeviationX1].Cmd.GoPoint_Condition[1]:=FALSE;	
END_IF

IF Mach_Control.U.DT_iMode=3 AND arrAxisCtrl[AxiseNo.AxisName.AndeviationX1].Status.Homed THEN
	arrAxisCtrl[AxiseNo.AxisName.AndeviationX1].Cmd.GoPoint_Condition[2]:=TRUE;
ELSE
	arrAxisCtrl[AxiseNo.AxisName.AndeviationX1].Cmd.GoPoint_Condition[2]:=FALSE;	
END_IF

IF Mach_Control.U.DT_iMode=3 AND arrAxisCtrl[AxiseNo.AxisName.AndeviationX1].Status.Homed THEN
	arrAxisCtrl[AxiseNo.AxisName.AndeviationX1].Cmd.GoPoint_Condition[3]:=TRUE;
ELSE
	arrAxisCtrl[AxiseNo.AxisName.AndeviationX1].Cmd.GoPoint_Condition[3]:=FALSE;	
END_IF

IF Mach_Control.U.DT_iMode=3 AND arrAxisCtrl[AxiseNo.AxisName.AndeviationX1].Status.Homed THEN
	arrAxisCtrl[AxiseNo.AxisName.AndeviationX1].Cmd.GoPoint_Condition[4]:=TRUE;
ELSE
	arrAxisCtrl[AxiseNo.AxisName.AndeviationX1].Cmd.GoPoint_Condition[4]:=FALSE;	
END_IF

IF Mach_Control.U.DT_iMode=3 AND arrAxisCtrl[AxiseNo.AxisName.AndeviationX1].Status.Homed THEN
	arrAxisCtrl[AxiseNo.AxisName.AndeviationX1].Cmd.GoPoint_Condition[5]:=TRUE;
ELSE
	arrAxisCtrl[AxiseNo.AxisName.AndeviationX1].Cmd.GoPoint_Condition[5]:=FALSE;	
END_IF

//正极纠偏平台X2
IF Mach_Control.U.DT_iMode=3  OR  (DP_Step0>=6015 AND   DP_Step0<=6041)   THEN
	arrAxisCtrl[AxiseNo.AxisName.AndeviationX2].Cmd.Home_Condition:=TRUE;
ELSE
	arrAxisCtrl[AxiseNo.AxisName.AndeviationX2].Cmd.Home_Condition:=FALSE;	
END_IF

IF Mach_Control.U.DT_iMode=3 AND arrAxisCtrl[AxiseNo.AxisName.AndeviationX2].Status.Homed THEN
	arrAxisCtrl[AxiseNo.AxisName.AndeviationX2].Cmd.GoPoint_Condition[1]:=TRUE;
ELSE
	arrAxisCtrl[AxiseNo.AxisName.AndeviationX2].Cmd.GoPoint_Condition[1]:=FALSE;	
END_IF

IF Mach_Control.U.DT_iMode=3 AND arrAxisCtrl[AxiseNo.AxisName.AndeviationX2].Status.Homed THEN
	arrAxisCtrl[AxiseNo.AxisName.AndeviationX2].Cmd.GoPoint_Condition[2]:=TRUE;
ELSE
	arrAxisCtrl[AxiseNo.AxisName.AndeviationX2].Cmd.GoPoint_Condition[2]:=FALSE;	
END_IF

IF Mach_Control.U.DT_iMode=3 AND arrAxisCtrl[AxiseNo.AxisName.AndeviationX2].Status.Homed THEN
	arrAxisCtrl[AxiseNo.AxisName.AndeviationX2].Cmd.GoPoint_Condition[3]:=TRUE;
ELSE
	arrAxisCtrl[AxiseNo.AxisName.AndeviationX2].Cmd.GoPoint_Condition[3]:=FALSE;	
END_IF

IF Mach_Control.U.DT_iMode=3 AND arrAxisCtrl[AxiseNo.AxisName.AndeviationX2].Status.Homed THEN
	arrAxisCtrl[AxiseNo.AxisName.AndeviationX2].Cmd.GoPoint_Condition[4]:=TRUE;
ELSE
	arrAxisCtrl[AxiseNo.AxisName.AndeviationX2].Cmd.GoPoint_Condition[4]:=FALSE;	
END_IF

IF Mach_Control.U.DT_iMode=3 AND arrAxisCtrl[AxiseNo.AxisName.AndeviationX2].Status.Homed THEN
	arrAxisCtrl[AxiseNo.AxisName.AndeviationX2].Cmd.GoPoint_Condition[5]:=TRUE;
ELSE
	arrAxisCtrl[AxiseNo.AxisName.AndeviationX2].Cmd.GoPoint_Condition[5]:=FALSE;	
END_IF

//正极纠偏平台Y
IF Mach_Control.U.DT_iMode=3  OR  (DP_Step0>=6015 AND   DP_Step0<=6041)   THEN
	arrAxisCtrl[AxiseNo.AxisName.AndeviationY].Cmd.Home_Condition:=TRUE;
ELSE
	arrAxisCtrl[AxiseNo.AxisName.AndeviationY].Cmd.Home_Condition:=FALSE;	
END_IF

IF Mach_Control.U.DT_iMode=3 AND arrAxisCtrl[AxiseNo.AxisName.AndeviationY].Status.Homed THEN
	arrAxisCtrl[AxiseNo.AxisName.AndeviationY].Cmd.GoPoint_Condition[1]:=TRUE;
ELSE
	arrAxisCtrl[AxiseNo.AxisName.AndeviationY].Cmd.GoPoint_Condition[1]:=FALSE;	
END_IF

IF Mach_Control.U.DT_iMode=3 AND arrAxisCtrl[AxiseNo.AxisName.AndeviationY].Status.Homed THEN
	arrAxisCtrl[AxiseNo.AxisName.AndeviationY].Cmd.GoPoint_Condition[2]:=TRUE;
ELSE
	arrAxisCtrl[AxiseNo.AxisName.AndeviationY].Cmd.GoPoint_Condition[2]:=FALSE;	
END_IF

IF Mach_Control.U.DT_iMode=3 AND arrAxisCtrl[AxiseNo.AxisName.AndeviationY].Status.Homed THEN
	arrAxisCtrl[AxiseNo.AxisName.AndeviationY].Cmd.GoPoint_Condition[3]:=TRUE;
ELSE
	arrAxisCtrl[AxiseNo.AxisName.AndeviationY].Cmd.GoPoint_Condition[3]:=FALSE;	
END_IF

IF Mach_Control.U.DT_iMode=3 AND arrAxisCtrl[AxiseNo.AxisName.AndeviationY].Status.Homed THEN
	arrAxisCtrl[AxiseNo.AxisName.AndeviationY].Cmd.GoPoint_Condition[4]:=TRUE;
ELSE
	arrAxisCtrl[AxiseNo.AxisName.AndeviationY].Cmd.GoPoint_Condition[4]:=FALSE;	
END_IF

IF Mach_Control.U.DT_iMode=3 AND arrAxisCtrl[AxiseNo.AxisName.AndeviationY].Status.Homed THEN
	arrAxisCtrl[AxiseNo.AxisName.AndeviationY].Cmd.GoPoint_Condition[5]:=TRUE;
ELSE
	arrAxisCtrl[AxiseNo.AxisName.AndeviationY].Cmd.GoPoint_Condition[5]:=FALSE;	
END_IF

//正极叠台搬运平移1
IF Mach_Control.U.DT_iMode=3 AND arrAxisCtrl[AxiseNo.AxisName.AnDTCarryingUpDown].Status.Homed AND
	arrAxisCtrl[AxiseNo.AxisName.AnDTCarryingUpDown].Status.fSetPos<= arrAxisPar[AxiseNo.AxisName.AnDTCarryingUpDown].arrTargetPoint[4]+1 AND
	arrAxisCtrl[AxiseNo.AxisName.AnCarryingLine].Status.fSetPos<=arrAxisPar[AxiseNo.AxisName.AnCarryingLine].arrTargetPoint[1] AND 
	arrCyCtrl[arrCyNo.CylinderName.AnScrapbinCy].Io.DIOnSwitch  AND NOT arrCyCtrl[arrCyNo.CylinderName.AnScrapbinCy].Io.DIOFFSwitch AND
	arrAxisCtrl[AxiseNo.AxisName.AnCarryingLine].Status.Homed AND arrAxisCtrl[AxiseNo.AxisName.AnCarryingLine].Status.NoMoving THEN
	arrAxisCtrl[AxiseNo.AxisName.AnDTCarryingLine].Cmd.Home_Condition:=TRUE;
ELSE
	arrAxisCtrl[AxiseNo.AxisName.AnDTCarryingLine].Cmd.Home_Condition:=FALSE;	
END_IF

IF Mach_Control.U.DT_iMode=3 AND arrCyCtrl[arrCyNo.CylinderName.AnScrapbinCy].Status.ONState THEN
   arrAxisCtrl[AxiseNo.AxisName.AnDTCarryingLine].Cmd.JogP_Condition:=TRUE;
   arrAxisCtrl[AxiseNo.AxisName.AnDTCarryingLine].Cmd.JogN_Condition:=TRUE;
   ELSE 
   arrAxisCtrl[AxiseNo.AxisName.AnDTCarryingLine].Cmd.JogP_Condition:=FALSE;
   arrAxisCtrl[AxiseNo.AxisName.AnDTCarryingLine].Cmd.JogN_Condition:=FALSE;
 END_IF

IF Mach_Control.U.DT_iMode=3 AND arrAxisCtrl[AxiseNo.AxisName.AnDTCarryingUpDown].Status.Homed AND
	arrAxisCtrl[AxiseNo.AxisName.AnDTCarryingUpDown].Status.fSetPos<= arrAxisPar[AxiseNo.AxisName.AnDTCarryingUpDown].arrTargetPoint[4]+1 AND
	arrAxisCtrl[AxiseNo.AxisName.AnCarryingLine].Cmd.arrbRealPoint[1] AND arrCyCtrl[arrCyNo.CylinderName.AnScrapbinCy].Status.ONState  THEN
	arrAxisCtrl[AxiseNo.AxisName.AnDTCarryingLine].Cmd.GoPoint_Condition[1]:=TRUE;
ELSE
	arrAxisCtrl[AxiseNo.AxisName.AnDTCarryingLine].Cmd.GoPoint_Condition[1]:=FALSE;	
END_IF

IF Mach_Control.U.DT_iMode=3 AND arrAxisCtrl[AxiseNo.AxisName.AnDTCarryingUpDown].Status.Homed AND
	arrAxisCtrl[AxiseNo.AxisName.AnDTCarryingUpDown].Status.fSetPos<= arrAxisPar[AxiseNo.AxisName.AnDTCarryingUpDown].arrTargetPoint[4]+1 AND
 	arrAxisCtrl[AxiseNo.AxisName.AnDTCarryingLine].Status.Homed AND arrAxisCtrl[AxiseNo.AxisName.SEPTATLine].Cmd.arrbRealPoint[2] AND
    arrCyCtrl[arrCyNo.CylinderName.AnScrapbinCy].Status.ONState THEN
	arrAxisCtrl[AxiseNo.AxisName.AnDTCarryingLine].Cmd.GoPoint_Condition[2]:=TRUE;
ELSE
	arrAxisCtrl[AxiseNo.AxisName.AnDTCarryingLine].Cmd.GoPoint_Condition[2]:=FALSE;	
END_IF


//正极叠台搬运升降1
IF Mach_Control.U.DT_iMode=3  THEN
	arrAxisCtrl[AxiseNo.AxisName.AnDTCarryingUpDown].Cmd.Home_Condition:=TRUE;
ELSE
	arrAxisCtrl[AxiseNo.AxisName.AnDTCarryingUpDown].Cmd.Home_Condition:=FALSE;	
END_IF

IF Mach_Control.U.DT_iMode=3 AND arrAxisCtrl[AxiseNo.AxisName.AnDTCarryingUpDown].Status.Homed THEN
	arrAxisCtrl[AxiseNo.AxisName.AnDTCarryingUpDown].Cmd.GoPoint_Condition[1]:=TRUE;
ELSE
	arrAxisCtrl[AxiseNo.AxisName.AnDTCarryingUpDown].Cmd.GoPoint_Condition[1]:=FALSE;	
END_IF

IF Mach_Control.U.DT_iMode=3 AND  arrAxisCtrl[AxiseNo.AxisName.AnDTCarryingUpDown].Status.Homed THEN
	arrAxisCtrl[AxiseNo.AxisName.AnDTCarryingUpDown].Cmd.GoPoint_Condition[2]:=TRUE;
ELSE
	arrAxisCtrl[AxiseNo.AxisName.AnDTCarryingUpDown].Cmd.GoPoint_Condition[2]:=FALSE;	
END_IF

IF Mach_Control.U.DT_iMode=3 AND arrAxisCtrl[AxiseNo.AxisName.AnDTCarryingUpDown].Status.Homed THEN
	arrAxisCtrl[AxiseNo.AxisName.AnDTCarryingUpDown].Cmd.GoPoint_Condition[3]:=TRUE;
ELSE
	arrAxisCtrl[AxiseNo.AxisName.AnDTCarryingUpDown].Cmd.GoPoint_Condition[3]:=FALSE;	
END_IF

IF Mach_Control.U.DT_iMode=3 AND arrAxisCtrl[AxiseNo.AxisName.AnDTCarryingUpDown].Status.Homed THEN
	arrAxisCtrl[AxiseNo.AxisName.AnDTCarryingUpDown].Cmd.GoPoint_Condition[4]:=TRUE;
ELSE
	arrAxisCtrl[AxiseNo.AxisName.AnDTCarryingUpDown].Cmd.GoPoint_Condition[4]:=FALSE;	
END_IF

IF Mach_Control.U.DT_iMode=3 AND arrAxisCtrl[AxiseNo.AxisName.AnDTCarryingUpDown].Status.Homed THEN
	arrAxisCtrl[AxiseNo.AxisName.AnDTCarryingUpDown].Cmd.GoPoint_Condition[5]:=TRUE;
ELSE
	arrAxisCtrl[AxiseNo.AxisName.AnDTCarryingUpDown].Cmd.GoPoint_Condition[5]:=FALSE;	
END_IF
//正极NG料盒伸缩气缸条件
IF arrAxisCtrl[AxiseNo.AxisName.AnDTCarryingUpDown].Cmd.arrbRealPoint[5] (*AND arrAxisCtrl[AxiseNo.AxisName.AnCarryingLine].Cmd.arrbRealPoint[1]*)  THEN
	arrCyCtrl[arrCyNo.CylinderName.	AnScrapbinCy].Cmd.OnCondition:=TRUE;
    arrCyCtrl[arrCyNo.CylinderName.	AnScrapbinCy].Cmd.OffCondition:=TRUE;
ELSE	
	arrCyCtrl[arrCyNo.CylinderName.	AnScrapbinCy].Cmd.OnCondition:=FALSE;
    arrCyCtrl[arrCyNo.CylinderName.	AnScrapbinCy].Cmd.OffCondition:=FALSE;	
END_IF
END_ACTION

ACTION An_Gohome:
An_GohomeTon(IN:= , PT:=T#1S , Q=> , ET=> );//正极取片回原点延时
An_GohomeOverTon(IN:= , PT:=T#90S , Q=> , ET=> );//负正回原点超时报警延时
rAn_Gohome_TRIG(CLK:=Mach_Control.An_b.An_GohomeHMI , Q=> );//正极取片回原点启动
fAn_Gohome_FRIG(CLK:=Mach_Control.An_b.An_GohomeHMI , Q=> );//负极回原点启动
//判断正极是否回原点完成
IF arrAxisCtrl[AxiseNo.AxisName.AnCarryingUpDown].Status.Homed AND  arrAxisCtrl[AxiseNo.AxisName.AnDTCarryingUpDown].Status.Homed  AND 
 	arrAxisCtrl[AxiseNo.AxisName.AnCarryingLine].Status.Homed AND arrAxisCtrl[AxiseNo.AxisName.AnCarryingWhirling].Status.Homed AND 				
	arrAxisCtrl[AxiseNo.AxisName.AndeviationX1].Status.Homed AND arrAxisCtrl[AxiseNo.AxisName.AndeviationX2].Status.Homed AND
	arrAxisCtrl[AxiseNo.AxisName.AndeviationY].Status.Homed	AND arrAxisCtrl[AxiseNo.AxisName.AnDTCarryingLine].Status.Homed AND An_GohomeDone THEN	
		Mach_Control.An_b.An_GohomeDone:=TRUE;//负极取片回原点完成
ELSE
		Mach_Control.An_b.An_GohomeDone:=FALSE;//负极取片回原点完成
END_IF




IF Mach_Control.U.DT_iMode=3 THEN//在手动状态下
		IF rAn_Gohome_TRIG.Q THEN
			Step_InitAnDT:=0;
			An_GohomeDone:=FALSE;
			An_Gohoming:=FALSE;//负极取片回原点中
			Mach_Control.An_b.An_GohomeDone:=FALSE;//负极取片回原点完成
		END_IF	
END_IF		
IF Mach_Control.U.DT_iMode=3 THEN//在手动状态下
	
//回原点超时报警	

IF  An_Gohoming THEN
		IF 	NOT An_GohomeOverTon.Q THEN
			    An_GohomeOverTon.IN:=TRUE;
		ELSE
			IF 	 An_GohomeOverTon.Q THEN
				An_Gohoming:=FALSE;
			     Mach_Control.An_b.Error[19]:=TRUE;//负极回原点超时报警
			     An_GohomeOverTon.IN:=FALSE;
			END_IF	 
				 
		END_IF

ELSE
		An_GohomeOverTon.IN:=FALSE;
END_IF




//正极取料机构初始C化
CASE Step_InitAnDT OF
0://等待正极回原点启动	
IF fAn_Gohome_FRIG.Q THEN
	An_Gohoming:=TRUE;//负极取片回原点中
	Mach_Control.An_b.An_GohomeHMI:=FALSE;
	Step_InitAnDT:=1;
END_IF
1://复位回原点完成
	An_GohomeDone:=FALSE;//正极回原点完成
	An_GohomeTon.IN:=FALSE;								
	IF NOT An_GohomeDone THEN
		Step_InitAnDT:=10;
	END_IF
10:
Mach_Control.An_b.An_CarryingFalg:=FALSE;//正极搬运升降有料标记
Mach_Control.An_b.An_DPCarryingFalg:=FALSE;//正极叠片搬运有料标记
Mach_Control.An_b.An_deviationFalg :=FALSE;//正极纠偏有料标记


An_StandbyStep0:=0;//正极纠偏平台自动步
An_StandbyStep1:=0;//正极取片备料步清零
An_StandbyStep2:=0;//叠正极片，判断真空、破真空
An_StandbyStep3:=0;//叠正极片，判断主轴是否完成
Mach_Control.An_b.AN_BeltDone:=FALSE;//取流水线取极片完成	
Mach_Control.An_b.An_MainBelting:=FALSE;// 复位正极搬运升降取极片中
An_Step0:=0;
An_Step1:=0;
An_Step2:=0;
An_Step3:=0;
An_StandbyStep0:=0;
An_Demarcate_Step0:=0;
An_RecdevPla_Step0:=0;						
Step_InitAnDT:=20;	
20:
	fbAnCamInCarryingLine.bCamInExecute:=FALSE;//正极送片搬运平移
	fbAnCamInCarryingUpDown.bCamInExecute:=FALSE;//正极送片搬运升降
	fbAnCamInCarryingWhirling.bCamInExecute:=FALSE;//正极送片搬运旋转
	fbAnCamInDTCarryingLine.bCamInExecute:=FALSE;//正极叠片搬运平移
	fbAnCamInDTCarryingUpDown.bCamInExecute:=FALSE;//正极叠片搬运升降
	IF NOT fbAnCamInCarryingLine.bCamInExecute AND NOT fbAnCamInCarryingUpDown.bCamInExecute AND 
		NOT  fbAnCamInCarryingWhirling.bCamInExecute AND NOT fbAnCamInDTCarryingLine.bCamInExecute AND 
		NOT  fbAnCamInDTCarryingUpDown.bCamInExecute THEN
				Step_InitAnDT:=25;	
	END_IF									
25:
arrAxisCtrl[AxiseNo.AxisName.AnCarryingUpDown].Cmd.bHalt:=TRUE;//正极送片搬运轴解耦
arrAxisCtrl[AxiseNo.AxisName.AnDTCarryingUpDown].Cmd.bHalt:=TRUE;//正极叠片搬运解耦
arrAxisCtrl[AxiseNo.AxisName.AnCarryingLine].Cmd.bHalt:=TRUE;//正极送片搬运平移轴解耦
arrAxisCtrl[AxiseNo.AxisName.AnDTCarryingLine].Cmd.bHalt:=TRUE;//正极叠片搬运平移轴解耦
arrAxisCtrl[AxiseNo.AxisName.AnCarryingWhirling].Cmd.bHalt:=TRUE;//正极送片搬运旋转轴解耦	
IF NOT arrAxisCtrl[AxiseNo.AxisName.AnCarryingUpDown].Status.Coupled AND arrAxisCtrl[AxiseNo.AxisName.AnCarryingUpDown].Status.NoMoving AND 
   NOT arrAxisCtrl[AxiseNo.AxisName.AnDTCarryingUpDown].Status.Coupled AND arrAxisCtrl[AxiseNo.AxisName.AnDTCarryingUpDown].Status.NoMoving AND
   NOT arrAxisCtrl[AxiseNo.AxisName.AnCarryingLine].Status.Coupled AND arrAxisCtrl[AxiseNo.AxisName.AnCarryingLine].Status.NoMoving AND 
   NOT arrAxisCtrl[AxiseNo.AxisName.AnDTCarryingLine].Status.Coupled AND arrAxisCtrl[AxiseNo.AxisName.AnDTCarryingLine].Status.NoMoving AND
   NOT arrAxisCtrl[AxiseNo.AxisName.AnCarryingWhirling].Status.Coupled AND arrAxisCtrl[AxiseNo.AxisName.AnCarryingWhirling].Status.NoMoving THEN
			arrAxisCtrl[AxiseNo.AxisName.AnCarryingUpDown].Cmd.bHalt:=FALSE;//正极送片搬运轴解耦
			arrAxisCtrl[AxiseNo.AxisName.AnDTCarryingUpDown].Cmd.bHalt:=FALSE;//正极叠片搬运解耦
			arrAxisCtrl[AxiseNo.AxisName.AnCarryingLine].Cmd.bHalt:=FALSE;//正极送片搬运平移轴解耦
			arrAxisCtrl[AxiseNo.AxisName.AnDTCarryingLine].Cmd.bHalt:=FALSE;//正极叠片搬运平移轴解耦
			arrAxisCtrl[AxiseNo.AxisName.AnCarryingWhirling].Cmd.bHalt:=FALSE;//正极送片搬运旋转轴解耦	
			Step_InitAnDT:=30;	
END_IF		
30:
arrAxisCtrl[AxiseNo.AxisName.AnCarryingUpDown].Cmd.bEnable:=TRUE;//正极送片搬运轴
arrAxisCtrl[AxiseNo.AxisName.AnDTCarryingUpDown].Cmd.bEnable:=TRUE;//正极叠片搬运
arrAxisCtrl[AxiseNo.AxisName.AnCarryingLine].Cmd.bEnable:=TRUE;//正极送片搬运平移轴
arrAxisCtrl[AxiseNo.AxisName.AnDTCarryingLine].Cmd.bEnable:=TRUE;//正极叠片搬运平移轴
arrAxisCtrl[AxiseNo.AxisName.AnCarryingWhirling].Cmd.bEnable:=TRUE;//正极送片搬运旋转轴	
arrAxisCtrl[AxiseNo.AxisName.AndeviationX1].Cmd.bEnable:=TRUE;//正极纠偏X1
arrAxisCtrl[AxiseNo.AxisName.AndeviationX2].Cmd.bEnable:=TRUE;//正极纠偏X2
arrAxisCtrl[AxiseNo.AxisName.AndeviationY].Cmd.bEnable:=TRUE;//正极纠偏Y						
IF arrAxisCtrl[AxiseNo.AxisName.AnCarryingUpDown].Status.Enabled AND 
   arrAxisCtrl[AxiseNo.AxisName.AnDTCarryingUpDown].Status.Enabled AND 
   arrAxisCtrl[AxiseNo.AxisName.AnCarryingLine].Status.Enabled AND 
   arrAxisCtrl[AxiseNo.AxisName.AnDTCarryingLine].Status.Enabled AND 
   arrAxisCtrl[AxiseNo.AxisName.AnCarryingWhirling].Status.Enabled AND
   arrAxisCtrl[AxiseNo.AxisName.AndeviationX1].Status.Enabled AND 
   arrAxisCtrl[AxiseNo.AxisName.AndeviationX2].Status.Enabled AND
   arrAxisCtrl[AxiseNo.AxisName.AndeviationY].Status.Enabled THEN
		Step_InitAnDT:=35;	
ELSIF arrAxisCtrl[AxiseNo.AxisName.AnCarryingUpDown].Status.Error OR 
   arrAxisCtrl[AxiseNo.AxisName.AnDTCarryingUpDown].Status.Error OR 
   arrAxisCtrl[AxiseNo.AxisName.AnCarryingLine].Status.Error OR 
   arrAxisCtrl[AxiseNo.AxisName.AnDTCarryingLine].Status.Error OR 
   arrAxisCtrl[AxiseNo.AxisName.AnCarryingWhirling].Status.Error OR
   arrAxisCtrl[AxiseNo.AxisName.AndeviationX1].Status.Error OR 
   arrAxisCtrl[AxiseNo.AxisName.AndeviationX2].Status.Error OR
   arrAxisCtrl[AxiseNo.AxisName.AndeviationY].Status.Error THEN
	An_Gohoming:=FALSE;//正极取片回原点中
		Step_InitAnDT:=9999;	
END_IF		

				
35://正极送片搬运升降、正极叠片搬运升降轴回原点
	arrAxisCtrl[AxiseNo.AxisName.AnCarryingUpDown].Cmd.bHome:=TRUE;//正极送片搬运轴回原点
	arrAxisCtrl[AxiseNo.AxisName.AnDTCarryingUpDown].Cmd.bHome:=TRUE;//正极叠片搬运回原点
	Step_InitAnDT:=40;
	
40://判断回原点是否完成
	IF NOT An_GohomeTon.Q THEN
			An_GohomeTon.IN:=TRUE;
	ELSE		
				IF arrAxisCtrl[AxiseNo.AxisName.AnCarryingUpDown].Status.Homed AND arrAxisCtrl[AxiseNo.AxisName.AnDTCarryingUpDown].Status.Homed  AND 
					arrAxisCtrl[AxiseNo.AxisName.AnCarryingUpDown].Status.NoMoving AND arrAxisCtrl[AxiseNo.AxisName.AnDTCarryingUpDown].Status.NoMoving  THEN
					arrAxisCtrl[AxiseNo.AxisName.AnCarryingUpDown].Cmd.bHome:=FALSE;//正极送片搬运轴回原点
					arrAxisCtrl[AxiseNo.AxisName.AnDTCarryingUpDown].Cmd.bHome:=FALSE;//正极叠片搬运回原点
					An_GohomeTon.IN:=FALSE;
					Step_InitAnDT:=45;
				ELSIF  arrAxisCtrl[AxiseNo.AxisName.AnCarryingUpDown].Status.Error OR arrAxisCtrl[AxiseNo.AxisName.AnDTCarryingUpDown].Status.Error THEN
						arrAxisCtrl[AxiseNo.AxisName.AnCarryingUpDown].Cmd.bHome:=FALSE;//正极送片搬运轴回原点
						arrAxisCtrl[AxiseNo.AxisName.AnDTCarryingUpDown].Cmd.bHome:=FALSE;//正极叠片搬运回原点
						An_GohomeTon.IN:=FALSE;
						An_Gohoming:=FALSE;//正极取片回原点中
						Step_InitAnDT:=9999;	  
				END_IF
	END_IF
45:
	IF arrAxisCtrl[AxiseNo.AxisName.AnDTCarryingUpDown].Status.Homed AND arrAxisCtrl[AxiseNo.AxisName.AnDTCarryingUpDown].Status.NoMoving THEN
		IF arrAxisCtrl[AxiseNo.AxisName.AnDTCarryingUpDown].Cmd.arrbRealPoint[5]  THEN
			arrAxisCtrl[AxiseNo.AxisName.AnDTCarryingUpDown].Cmd.iGoSetPos:=0;
			Step_InitAnDT:=50;
		ELSE
		   arrAxisCtrl[AxiseNo.AxisName.AnDTCarryingUpDown].Cmd.iGoSetPos:=5;
		END_IF	
	END_IF		
	IF  arrAxisCtrl[AxiseNo.AxisName.AnDTCarryingUpDown].Status.Error THEN
		An_Gohoming:=FALSE;//正极取片回原点中
		Step_InitAnDT:=9999;
	END_IF		
	
50://NG料盒气缸伸出
IF arrAxisCtrl[AxiseNo.AxisName.AnDTCarryingUpDown].Cmd.arrbRealPoint[5] OR arrCyCtrl[arrCyNo.CylinderName.AnScrapbinCy].Io.DIOnSwitch THEN
	arrCyCtrl[arrCyNo.CylinderName.AnScrapbinCy].Cmd.bON:=TRUE;//正极纠偏气缸伸出
	IF  arrCyCtrl[arrCyNo.CylinderName.AnScrapbinCy].Status.ONState THEN
		Step_InitAnDT:=60;	
	ELSIF arrCyCtrl[arrCyNo.CylinderName.AnScrapbinCy].Status.Error1 OR  arrCyCtrl[arrCyNo.CylinderName.AnScrapbinCy].Status.Error2 THEN
		An_Gohoming:=FALSE;//正极取片回原点中
		Step_InitAnDT:=9999;
	END_IF	
ELSE
	Mach_Control.An_b.Error[41] :=TRUE;//正极机械手初始化时，叠台搬运升降不在避让位
	An_Gohoming:=FALSE;//正极取片回原点中
	Step_InitAnDT:=9999;
END_IF	
	
60://正极送片搬运平移、叠片搬运平移、送片搬运旋转轴回原点、正极纠偏X1、正极纠偏X2、正极纠偏Y回原点
	arrAxisCtrl[AxiseNo.AxisName.AnCarryingLine].Cmd.bHome:=TRUE;//正极送片搬运平移轴回原点
	//arrAxisCtrl[AxiseNo.AxisName.AnCarryingWhirling].Cmd.bHome:=TRUE;//正极送片搬运旋转轴回原点								
	arrAxisCtrl[AxiseNo.AxisName.AndeviationX1].Cmd.bHome:=TRUE;//正极纠偏X1
	arrAxisCtrl[AxiseNo.AxisName.AndeviationX2].Cmd.bHome:=TRUE;//正极纠偏X2				
	arrAxisCtrl[AxiseNo.AxisName.AndeviationY].Cmd.bHome:=TRUE;//正极纠偏Y	
	An_CarryingTorMark:=TRUE;//正极搬运1移位力矩判断标志位									
	Step_InitAnDT:=70;
70://判断正极送片搬运平移、叠片搬运平移、送片搬运旋转回原点是否完成
	IF NOT An_GohomeTon.Q THEN		
		An_GohomeTon.IN:=TRUE;
	ELSE		
		IF arrAxisCtrl[AxiseNo.AxisName.AnCarryingLine].Status.Homed AND arrAxisCtrl[AxiseNo.AxisName.AnCarryingLine].Status.NoMoving (*AND
		 arrAxisCtrl[AxiseNo.AxisName.AnCarryingWhirling].Status.Homed*) AND  arrAxisCtrl[AxiseNo.AxisName.AnCarryingWhirling].Status.NoMoving  AND   						
		arrAxisCtrl[AxiseNo.AxisName.AndeviationX1].Status.Homed AND arrAxisCtrl[AxiseNo.AxisName.AndeviationX1].Status.NoMoving AND 
		arrAxisCtrl[AxiseNo.AxisName.AndeviationX2].Status.Homed AND arrAxisCtrl[AxiseNo.AxisName.AndeviationX2].Status.NoMoving AND
			arrAxisCtrl[AxiseNo.AxisName.AndeviationY].Status.Homed AND arrAxisCtrl[AxiseNo.AxisName.AndeviationY].Status.NoMoving   THEN
			arrAxisCtrl[AxiseNo.AxisName.AnCarryingLine].Cmd.bHome:=FALSE;//正极送片搬运平移轴回原点
			arrAxisCtrl[AxiseNo.AxisName.AnDTCarryingLine].Cmd.bHome:=FALSE;//正极叠片搬运平移轴回原点
			arrAxisCtrl[AxiseNo.AxisName.AnCarryingWhirling].Cmd.bHome:=FALSE;//正极送片搬运旋转轴回原点		
			arrAxisCtrl[AxiseNo.AxisName.AndeviationX1].Cmd.bHome:=FALSE;//正极纠偏X1		
			arrAxisCtrl[AxiseNo.AxisName.AndeviationX2].Cmd.bHome:=FALSE;//正极纠偏X2
			arrAxisCtrl[AxiseNo.AxisName.AndeviationY].Cmd.bHome:=FALSE;//正极纠偏Y
			An_CarryingTorMark:=FALSE;//正极搬运1移位力矩判断标志位			
			An_GohomeTon.IN:=FALSE;
			Step_InitAnDT:=75;
		ELSIF arrAxisCtrl[AxiseNo.AxisName.AnCarryingLine].Status.Error OR arrAxisCtrl[AxiseNo.AxisName.AnCarryingWhirling].Status.Error OR				
			arrAxisCtrl[AxiseNo.AxisName.AndeviationX1].Status.Error OR arrAxisCtrl[AxiseNo.AxisName.AndeviationX2].Status.Error OR 
			arrAxisCtrl[AxiseNo.AxisName.AndeviationY].Status.Error THEN
			arrAxisCtrl[AxiseNo.AxisName.AnCarryingLine].Cmd.bHome:=FALSE;//正极送片搬运平移轴回原点
			arrAxisCtrl[AxiseNo.AxisName.AnDTCarryingLine].Cmd.bHome:=FALSE;//正极叠片搬运平移轴回原点
			arrAxisCtrl[AxiseNo.AxisName.AnCarryingWhirling].Cmd.bHome:=FALSE;//正极送片搬运旋转轴回原点		
			arrAxisCtrl[AxiseNo.AxisName.AndeviationX1].Cmd.bHome:=FALSE;//正极纠偏X1		
			arrAxisCtrl[AxiseNo.AxisName.AndeviationX2].Cmd.bHome:=FALSE;//正极纠偏X2
			arrAxisCtrl[AxiseNo.AxisName.AndeviationY].Cmd.bHome:=FALSE;//正极纠偏Y
			An_GohomeTon.IN:=FALSE;
			An_Gohoming:=FALSE;//正极取片回原点中
			Step_InitAnDT:=9999;
		END_IF
	END_IF
75:
	//极送片搬运平移轴移动至初始位
	IF arrAxisCtrl[AxiseNo.AxisName.AnCarryingLine].Status.Homed AND arrAxisCtrl[AxiseNo.AxisName.AnCarryingLine].Status.NoMoving THEN
		IF arrAxisCtrl[AxiseNo.AxisName.AnCarryingLine].Cmd.arrbRealPoint[1] THEN
		   arrAxisCtrl[AxiseNo.AxisName.AnCarryingLine].Cmd.iGoSetPos:=0;
		 ELSE
			arrAxisCtrl[AxiseNo.AxisName.AnCarryingLine].Cmd.iGoSetPos:=1; 
		END_IF	
	END_IF
	(*//正极送片搬运旋转轴移动至初始位
	IF arrAxisCtrl[AxiseNo.AxisName.AnCarryingWhirling].Status.Homed AND arrAxisCtrl[AxiseNo.AxisName.AnCarryingWhirling].Status.NoMoving THEN
		IF arrAxisCtrl[AxiseNo.AxisName.AnCarryingWhirling].Cmd.arrbRealPoint[1]  THEN
			arrAxisCtrl[AxiseNo.AxisName.AnCarryingWhirling].Cmd.iGoSetPos:=0;
		ELSE
		   arrAxisCtrl[AxiseNo.AxisName.AnCarryingWhirling].Cmd.iGoSetPos:=1;
		END_IF
	END_IF*)
	//正极纠偏X1
	IF arrAxisCtrl[AxiseNo.AxisName.AndeviationX1].Status.Homed AND arrAxisCtrl[AxiseNo.AxisName.AndeviationX1].Status.NoMoving THEN
		IF arrAxisCtrl[AxiseNo.AxisName.AndeviationX1].Cmd.arrbRealPoint[1]  THEN
			arrAxisCtrl[AxiseNo.AxisName.AndeviationX1].Cmd.iGoSetPos:=0;
		ELSE
		   arrAxisCtrl[AxiseNo.AxisName.AndeviationX1].Cmd.iGoSetPos:=1;
		END_IF
	END_IF
	//正极纠偏X2
	IF arrAxisCtrl[AxiseNo.AxisName.AndeviationX2].Status.Homed AND arrAxisCtrl[AxiseNo.AxisName.AndeviationX2].Status.NoMoving THEN
		IF arrAxisCtrl[AxiseNo.AxisName.AndeviationX2].Cmd.arrbRealPoint[1]  THEN
			arrAxisCtrl[AxiseNo.AxisName.AndeviationX2].Cmd.iGoSetPos:=0;
		ELSE
		   arrAxisCtrl[AxiseNo.AxisName.AndeviationX2].Cmd.iGoSetPos:=1;
		END_IF
	END_IF	
	//正极纠偏Y
	IF arrAxisCtrl[AxiseNo.AxisName.AndeviationY].Status.Homed AND arrAxisCtrl[AxiseNo.AxisName.AndeviationY].Status.NoMoving THEN
		IF arrAxisCtrl[AxiseNo.AxisName.AndeviationY].Cmd.arrbRealPoint[1]  THEN
			arrAxisCtrl[AxiseNo.AxisName.AndeviationY].Cmd.iGoSetPos:=0;
		ELSE
		   arrAxisCtrl[AxiseNo.AxisName.AndeviationY].Cmd.iGoSetPos:=1;
		END_IF
	END_IF								
	
	IF 	arrAxisCtrl[AxiseNo.AxisName.AnCarryingLine].Cmd.arrbRealPoint[1] AND arrAxisCtrl[AxiseNo.AxisName.AnCarryingLine].Status.NoMoving AND
		(*arrAxisCtrl[AxiseNo.AxisName.AnCarryingWhirling].Cmd.arrbRealPoint[1] AND *)arrAxisCtrl[AxiseNo.AxisName.AnCarryingWhirling].Status.NoMoving AND
		arrAxisCtrl[AxiseNo.AxisName.AndeviationX1].Cmd.arrbRealPoint[1]  AND arrAxisCtrl[AxiseNo.AxisName.AndeviationX1].Status.NoMoving AND
		arrAxisCtrl[AxiseNo.AxisName.AndeviationX2].Cmd.arrbRealPoint[1] AND arrAxisCtrl[AxiseNo.AxisName.AndeviationX2].Status.NoMoving AND
		arrAxisCtrl[AxiseNo.AxisName.AndeviationY].Cmd.arrbRealPoint[1]	 AND	arrAxisCtrl[AxiseNo.AxisName.AndeviationY].Status.NoMoving THEN
					Step_InitAnDT:=80;
					arrAxisCtrl[AxiseNo.AxisName.AnCarryingWhirling].Cmd.bHome:=TRUE;//正极送片搬运旋转轴回原点
					
	ELSIF  arrAxisCtrl[AxiseNo.AxisName.AnCarryingLine].Status.Error AND arrAxisCtrl[AxiseNo.AxisName.AnCarryingWhirling].Status.Error AND
		arrAxisCtrl[AxiseNo.AxisName.AndeviationX1].Status.Error AND arrAxisCtrl[AxiseNo.AxisName.AndeviationX2].Status.Error AND 
		arrAxisCtrl[AxiseNo.AxisName.AndeviationY].Status.Error THEN
		An_Gohoming:=FALSE;//正极取片回原点中
		Step_InitAnDT:=9999;
	END_IF	
80://正极送片搬运旋转轴回原点	
IF  arrAxisCtrl[AxiseNo.AxisName.AnCarryingWhirling].Status.Homed		THEN
	arrAxisCtrl[AxiseNo.AxisName.AnCarryingWhirling].Cmd.bHome:=FALSE;//正极送片搬运旋转轴回原点	
	Step_InitAnDT:=83;	
END_IF			

83://正极送片搬运旋转轴移动至初始位
	IF arrAxisCtrl[AxiseNo.AxisName.AnCarryingWhirling].Status.Homed AND arrAxisCtrl[AxiseNo.AxisName.AnCarryingWhirling].Status.NoMoving THEN
		IF arrAxisCtrl[AxiseNo.AxisName.AnCarryingWhirling].Cmd.arrbRealPoint[1]  THEN
			arrAxisCtrl[AxiseNo.AxisName.AnCarryingWhirling].Cmd.iGoSetPos:=0;
			Step_InitAnDT:=85;
		ELSE
		   arrAxisCtrl[AxiseNo.AxisName.AnCarryingWhirling].Cmd.iGoSetPos:=1;
		END_IF
	END_IF

85://叠片搬运回原点							
	arrAxisCtrl[AxiseNo.AxisName.AnDTCarryingLine].Cmd.bHome:=TRUE;//正极叠片搬运平移轴回原点
	An_DTCarryingTorMark:=TRUE;//正极叠台搬运力矩判断标志位	
	Step_InitAnDT:=90;	
90://判断叠片搬运回原点是否完成
	IF NOT An_GohomeTon.Q THEN
		An_GohomeTon.IN:=TRUE;
	ELSE
		IF arrAxisCtrl[AxiseNo.AxisName.AnDTCarryingLine].Status.Homed AND arrAxisCtrl[AxiseNo.AxisName.AnDTCarryingLine].Status.NoMoving  THEN
			An_GohomeTon.IN:=FALSE;	
			arrAxisCtrl[AxiseNo.AxisName.AnDTCarryingLine].Cmd.bHome:=FALSE;//正极叠片搬运平移轴回原点
			An_DTCarryingTorMark:=FALSE;//正极叠台搬运力矩判断标志位	
			Step_InitAnDT:=100;
		ELSIF arrAxisCtrl[AxiseNo.AxisName.AnDTCarryingLine].Status.Error THEN
			An_GohomeTon.IN:=FALSE;	
			arrAxisCtrl[AxiseNo.AxisName.AnDTCarryingLine].Cmd.bHome:=FALSE;//正极叠片搬运平移轴回原点
		    An_Gohoming:=FALSE;//正极取片回原点中
			Step_InitAnDT:=9999;
		END_IF
	END_IF
100://轴移动到初始位置	
	//正极叠片搬运平移轴移动至初始位
	IF arrAxisCtrl[AxiseNo.AxisName.AnDTCarryingLine].Status.Homed AND arrAxisCtrl[AxiseNo.AxisName.AnDTCarryingLine].Status.NoMoving THEN
		IF arrAxisCtrl[AxiseNo.AxisName.AnDTCarryingLine].Cmd.arrbRealPoint[1]  THEN
			arrAxisCtrl[AxiseNo.AxisName.AnDTCarryingLine].Cmd.iGoSetPos:=0;
			Step_InitAnDT:=110;
		ELSE
		   arrAxisCtrl[AxiseNo.AxisName.AnDTCarryingLine].Cmd.iGoSetPos:=1;
		END_IF	
	ELSIF arrAxisCtrl[AxiseNo.AxisName.AnDTCarryingLine].Status.Error THEN
		An_Gohoming:=FALSE;//正极取片回原点中
		Step_InitAnDT:=9999;
	END_IF
110:
	arrCyCtrl[arrCyNo.ElectValveName.AnCarryingVacuum].Cmd.bOFF:=TRUE;//正极搬运升降取料真空关
	arrCyCtrl[arrCyNo.ElectValveName.AnCarryingVacuum].Cmd.bON:=FALSE;//正极搬运升降取料真空关
	
	arrCyCtrl[arrCyNo.ElectValveName.AnCarryingVacuumBark].Cmd.bOFF:=TRUE;//正极搬运升降取料破真空关
	arrCyCtrl[arrCyNo.ElectValveName.AnCarryingVacuumBark].Cmd.bON:=FALSE;//正极搬运升降取料破真空关
	
	arrCyCtrl[arrCyNo.ElectValveName.AndeviationVacuum].Cmd.bOFF:=TRUE;//正极纠偏平台真空关
	arrCyCtrl[arrCyNo.ElectValveName.AndeviationVacuum].Cmd.bON:=FALSE;//正极纠偏平台真空关
	
	arrCyCtrl[arrCyNo.ElectValveName.AndeviationVacuumBark].Cmd.bOFF:=TRUE;//正极纠偏平台破真空关
	arrCyCtrl[arrCyNo.ElectValveName.AndeviationVacuumBark].Cmd.bON:=FALSE;//正极纠偏平台破真空关
	
	arrCyCtrl[arrCyNo.ElectValveName.AnDTCarryingVacuum].Cmd.bOFF:=FALSE;//正极叠片搬运真空关
	arrCyCtrl[arrCyNo.ElectValveName.AnDTCarryingVacuum].Cmd.bON:=TRUE;//正极叠片搬运真空关
	
	arrCyCtrl[arrCyNo.ElectValveName.AnDTCarryingVacuumBark].Cmd.bON:=TRUE;//正极叠片搬运破真空关	
	arrCyCtrl[arrCyNo.ElectValveName.AnDTCarryingVacuumBark].Cmd.bOFF:=FALSE;//正极叠片搬运破真空关				
	//正极送片搬运升降移动至等待位
	IF arrAxisCtrl[AxiseNo.AxisName.AnCarryingUpDown].Status.Homed AND arrAxisCtrl[AxiseNo.AxisName.AnCarryingUpDown].Status.NoMoving THEN
		IF arrAxisCtrl[AxiseNo.AxisName.AnCarryingUpDown].Cmd.arrbRealPoint[4] THEN
		   arrAxisCtrl[AxiseNo.AxisName.AnCarryingUpDown].Cmd.iGoSetPos:=0;
		 ELSE
			arrAxisCtrl[AxiseNo.AxisName.AnCarryingUpDown].Cmd.iGoSetPos:=4;
		END_IF
	END_IF
	//正极叠片搬运升降移动至等待位
	IF arrAxisCtrl[AxiseNo.AxisName.AnDTCarryingUpDown].Status.Homed AND arrAxisCtrl[AxiseNo.AxisName.AnDTCarryingUpDown].Status.NoMoving THEN
		IF  arrAxisCtrl[AxiseNo.AxisName.AnDTCarryingUpDown].Cmd.arrbRealPoint[4] THEN
				arrAxisCtrl[AxiseNo.AxisName.AnDTCarryingUpDown].Cmd.iGoSetPos:=0;
		 ELSE
				arrAxisCtrl[AxiseNo.AxisName.AnDTCarryingUpDown].Cmd.iGoSetPos:=4;
		END_IF	
	END_IF		
	IF  	arrAxisCtrl[AxiseNo.AxisName.AnCarryingUpDown].Cmd.arrbRealPoint[4] AND arrAxisCtrl[AxiseNo.AxisName.AnCarryingUpDown].Status.NoMoving  AND 
		arrAxisCtrl[AxiseNo.AxisName.AnDTCarryingUpDown].Cmd.arrbRealPoint[4] AND 	arrAxisCtrl[AxiseNo.AxisName.AnDTCarryingUpDown].Status.NoMoving  THEN
		An_GohomeDone:=TRUE;//正极回原点完成
		An_Gohoming:=FALSE;//正极取片回原点中
		Step_InitAnDT:=0;
	ELSIF arrAxisCtrl[AxiseNo.AxisName.AnCarryingUpDown].Status.Error OR arrAxisCtrl[AxiseNo.AxisName.AnDTCarryingUpDown].Status.Error THEN
		An_Gohoming:=FALSE;//正极取片回原点中
		Step_InitAnDT:=9999;
	END_IF
END_CASE
END_IF
END_ACTION

ACTION An_OverNG:
DT_TON[1](IN:= , PT:=T#300MS , Q=> , ET=> );//
DT_TON[2](IN:= , PT:=T#300MS , Q=> , ET=> );//
DT_TON[3](IN:= , PT:=T#200MS , Q=> , ET=> );//
DT_TON[4](IN:= , PT:=T#200MS , Q=> , ET=> );//
(*******************************************************************************************************踢正极对齐度NG片**************************************************************************************************************************)
 IF   An_OverNGStep=1630 THEN
	arrAxisCtrl[AxiseNo.AxisName.AnDTCarryingUpDown].Cmd.fOverride:=50;
 ELSE
   arrAxisCtrl[AxiseNo.AxisName.AnDTCarryingUpDown].Cmd.fOverride:=100;
 END_IF
 

 
 IF  AnOverNGcount>=3 OR CaOverNGcount>=3 THEN
     OversequelNG:=TRUE;	
 END_IF
 
IF Mach_Control.U.DT_iMode=1 THEN//在自动状态下
   CASE An_OverNGStep OF   
			1000://判断正极叠台搬运是否有片，有片的话放到纠偏台
						fAnScaling:=1;//20240508 CF
		            	fCaScaling:=1;//20240508 CF		
						AnOverNGcount:=AnOverNGcount+1;
						IF arrCyCtrl[arrCyNo.ElectValveName.AnDTCarryingVacuum].Io.DIOnSwitch AND  Mach_Control.An_b.An_DPCarryingFalg  THEN//正极再取片位且叠台搬运有片,把当前片放到纠偏台
							An_OverNGStep:=1010;
						ELSE
							An_OverNGStep:=1050;	
						END_IF
	
			1010://纠偏台回初始位
				//纠偏平台X1移动至初始位
				IF NOT DP_SinStepe THEN
					IF arrAxisCtrl[AxiseNo.AxisName.AndeviationX1].Status.Homed  AND arrAxisCtrl[AxiseNo.AxisName.AndeviationX1].Status.NoMoving AND NOT  arrAxisCtrl[AxiseNo.AxisName.AndeviationX1].Status.Error THEN
						IF arrAxisCtrl[AxiseNo.AxisName.AndeviationX1].Cmd.arrbRealPoint[1] THEN
							arrAxisCtrl[AxiseNo.AxisName.AndeviationX1].Cmd.iGoSetPos:=0;
						ELSE
							arrAxisCtrl[AxiseNo.AxisName.AndeviationX1].Cmd.iGoSetPos:=1;
						END_IF					
					END_IF
					//纠偏平台X2移动至初始位
					IF arrAxisCtrl[AxiseNo.AxisName.AndeviationX2].Status.Homed  AND arrAxisCtrl[AxiseNo.AxisName.AndeviationX2].Status.NoMoving AND NOT  arrAxisCtrl[AxiseNo.AxisName.AndeviationX2].Status.Error THEN
						IF arrAxisCtrl[AxiseNo.AxisName.AndeviationX2].Cmd.arrbRealPoint[1] THEN
							arrAxisCtrl[AxiseNo.AxisName.AndeviationX2].Cmd.iGoSetPos:=0;
						ELSE
							arrAxisCtrl[AxiseNo.AxisName.AndeviationX2].Cmd.iGoSetPos:=1;
						END_IF					
					END_IF
					//纠偏平台X2移动至初始位
					IF arrAxisCtrl[AxiseNo.AxisName.AndeviationY].Status.Homed  AND arrAxisCtrl[AxiseNo.AxisName.AndeviationY].Status.NoMoving AND NOT  arrAxisCtrl[AxiseNo.AxisName.AndeviationY].Status.Error THEN
						IF arrAxisCtrl[AxiseNo.AxisName.AndeviationY].Cmd.arrbRealPoint[1] THEN
							arrAxisCtrl[AxiseNo.AxisName.AndeviationY].Cmd.iGoSetPos:=0;
						ELSE
							arrAxisCtrl[AxiseNo.AxisName.AndeviationY].Cmd.iGoSetPos:=1;
						END_IF					
					END_IF
					IF arrAxisCtrl[AxiseNo.AxisName.AndeviationX1].Cmd.arrbRealPoint[1] AND arrAxisCtrl[AxiseNo.AxisName.AndeviationX2].Cmd.arrbRealPoint[1] AND arrAxisCtrl[AxiseNo.AxisName.AndeviationY].Cmd.arrbRealPoint[1] THEN
						DT_SingeMode();//单步选择	
						An_OverNGStep:=1020;
                        DT_TON[3].IN:=FALSE; 	
					END_IF	
				END_IF
			1020://叠台搬运极片放回纠偏台
				IF NOT DP_SinStepe THEN
					IF arrAxisCtrl[AxiseNo.AxisName.AnDTCarryingLine].Cmd.arrbRealPoint[1]  AND NOT Mach_Control.An_b.An_deviationFalg THEN 
						IF arrAxisCtrl[AxiseNo.AxisName.AnDTCarryingUpDown].Cmd.arrbRealPoint[2] THEN
							arrAxisCtrl[AxiseNo.AxisName.AnDTCarryingUpDown].Cmd.iGoSetPos:=0;
					    ELSE
							arrAxisCtrl[AxiseNo.AxisName.AnDTCarryingUpDown].Cmd.iGoSetPos:=2;//正极叠台搬运下降至取片位
					    END_IF
                   END_IF
				       IF arrAxisCtrl[AxiseNo.AxisName.AnDTCarryingUpDown].Cmd.arrbRealPoint[2] THEN
				           	/// 吸盘破真空    纠偏台开真空
				
							arrCyCtrl[arrCyNo.ElectValveName.AnDTCarryingVacuum].Cmd.bOFF:=FALSE;//正极叠片搬运升降真空关
							arrCyCtrl[arrCyNo.ElectValveName.AnDTCarryingVacuum].Cmd.bON:=TRUE;//正极叠片搬运升降真空关
						
							arrCyCtrl[arrCyNo.ElectValveName.AndeviationVacuum].Cmd.bON:=TRUE;	//正极纠偏台真空			
							arrCyCtrl[arrCyNo.ElectValveName.AndeviationVacuum].Cmd.bOFF:=FALSE;	//正极纠偏台真空	   
							DT_SingeMode();//单步选择	
							An_OverNGStep:=1030;
							DT_TON[3].IN:=TRUE;
							Mach_Control.An_b.An_deviationFalg:=TRUE;//置位纠偏平台有料标记
						    Mach_Control.An_b.An_DPCarryingFalg:=FALSE;//正极搬运真空吸盘有料标记复位
	                    END_IF
				END_IF
			1030://叠台搬运极片上升至凸轮耦合初始高度
				IF NOT DP_SinStepe  AND DT_TON[3].Q THEN
					IF arrAxisCtrl[AxiseNo.AxisName.AnDTCarryingUpDown].Cmd.arrbRealPoint[4]  THEN
						arrAxisCtrl[AxiseNo.AxisName.AnDTCarryingUpDown].Cmd.iGoSetPos:=0;
						/// 吸盘破真空    纠偏台开真空
						Mach_Control.An_b.An_deviationFalg:=TRUE;//置位纠偏平台有料标记
						Mach_Control.An_b.An_DPCarryingFalg:=FALSE;//正极搬运真空吸盘有料标记复位
						Par.stDT_date.An_MQ_Slice[1]:=Par.stDT_date.An_MQ_Slice[2];
						DT_SingeMode();//单步选择	
						An_OverNGStep:=1050;
						DT_TON[3].IN:=FALSE;
					ELSE
						arrAxisCtrl[AxiseNo.AxisName.AnDTCarryingUpDown].Cmd.iGoSetPos:=4;//正极搬运升降2上升至凸轮耦合初始高度
					END_IF			
				END_IF		   
		
            1050://判断主轴是否停止、是否在初始位、是否有轴在耦合中
					IF NOT DP_SinStepe THEN
								IF arrAxis[AxiseNo.VirAxisName.VirMain].Status.NotMoving AND arrAxis[AxiseNo.VirAxisName.VirMain].NcToPlc.SetPos=0 AND NOT DT_AxiseCoupling THEN
									DT_SingeMode();//单步选择
									An_OverNGStep:=1070;
								ELSE
									DP_Step1:=100;//调用主轴回初始位子程序
									DT_SingeMode();//单步选择
									An_OverNGStep:=1060;
								END_IF
			    	END_IF		
			1060://判断主轴的模长的当前位置是否为0
				IF NOT DP_SinStepe THEN
					IF DP_Step1=6666 AND arrAxis[AxiseNo.VirAxisName.VirMain].Status.NotMoving AND arrAxis[AxiseNo.VirAxisName.VirMain].NcToPlc.SetPos=0 AND NOT DT_AxiseCoupling  THEN
						DT_SingeMode();//单步选择
						An_OverNGStep:=1070;
					END_IF	
				END_IF							

			1070://判断NG气缸是否在安全位
					IF arrCyCtrl[arrCyNo.CylinderName.AnScrapbinCy].Status.ONState AND arrCyCtrl[arrCyNo.CylinderName.CaScrapbinUDCy].Status.OFFState AND
						arrCyCtrl[arrCyNo.CylinderName.AnScrapbinCy].Status.ONState AND arrCyCtrl[arrCyNo.CylinderName.PreDiaph].Status.OFFState AND 
						arrCyCtrl[arrCyNo.CylinderName.PoleHotCutterCy].Status.OFFState AND arrCyCtrl[arrCyNo.CylinderName.PoleTapeCy].Status.OFFState AND
						arrCyCtrl[arrCyNo.CylinderName.PoleTapeSplicerRCy].Status.ONState AND arrCyCtrl[arrCyNo.CylinderName.PoleTapeSplicerLCy].Status.ONState AND 
                        arrAxisCtrl[AxiseNo.AxisName.LeftYDUpDown].Cmd.arrbRealPoint[1] AND arrAxisCtrl[AxiseNo.AxisName.RightYDUpDown].Cmd.arrbRealPoint[1]    THEN
						An_OverNGStep:=1100;		
					ELSE
						An_OverNGStep:=1080;	
					END_IF
			1080:
						arrCyCtrl[arrCyNo.CylinderName.AnScrapbinCy].Cmd.bON:=TRUE;
						arrCyCtrl[arrCyNo.CylinderName.PreDiaph].Cmd.bOFF:=TRUE;
						arrCyCtrl[arrCyNo.CylinderName.PoleHotCutterCy].Cmd.bOFF:=TRUE;
						arrCyCtrl[arrCyNo.CylinderName.PoleTapeCy].Cmd.bOFF:=TRUE;
						arrCyCtrl[arrCyNo.CylinderName.PoleTapeSplicerRCy].Cmd.bON:=TRUE;
						arrCyCtrl[arrCyNo.CylinderName.PoleTapeSplicerLCy].Cmd.bON:=TRUE;
						arrCyCtrl[arrCyNo.CylinderName.AnScrapbinCy].Cmd.bON:=TRUE;
						IF   arrCyCtrl[arrCyNo.CylinderName.AnScrapbinCy].Status.ONState AND  arrCyCtrl[arrCyNo.CylinderName.PreDiaph].Status.OFFState AND 
							arrCyCtrl[arrCyNo.CylinderName.PoleHotCutterCy].Status.OFFState AND arrCyCtrl[arrCyNo.CylinderName.PoleTapeCy].Status.OFFState AND
							arrCyCtrl[arrCyNo.CylinderName.PoleTapeSplicerRCy].Status.ONState AND arrCyCtrl[arrCyNo.CylinderName.PoleTapeSplicerLCy].Status.ONState THEN
							An_OverNGStep:=1090;									
						END_IF
			1090:
					arrCyCtrl[arrCyNo.CylinderName.CaScrapbinUDCy].Cmd.bOFF:=TRUE;
					IF  arrCyCtrl[arrCyNo.CylinderName.CaScrapbinUDCy].Status.OFFState AND  arrAxisCtrl[AxiseNo.AxisName.LeftYDUpDown].Cmd.arrbRealPoint[1] 
                         AND arrAxisCtrl[AxiseNo.AxisName.RightYDUpDown].Cmd.arrbRealPoint[1] THEN
						An_OverNGStep:=1100;	
					END_IF	

              1100:
						IF NOT DP_SinStepe AND TailCurlSEPTA_SafePos THEN		
									Scan_TON[2].IN:=TRUE;	
										IF 	An_CarryingPos1  THEN//正极搬运、叠片各轴在初始位
											         Scan_TON[1].IN:=TRUE;	
													 DTPosError[11]:=FALSE;
													 IF CA_CarryingPos2  THEN//负极在叠片位	
														             DTPosError[12]:=FALSE;
																IF arrAxisCtrl[AxiseNo.AxisName.SEPTATLine].Cmd.arrbRealPoint[1]   THEN													
																	DT_SingeMode();//单步选择											
																	An_OverNGStep:=1200;//													
																ELSE
																	Mach_Control.DT_b.Error[6]:=TRUE;//叠正极片凸轮耦合时，隔膜平移轴即不在正极叠片位，也不在正极叠片位报警
																//	An_OverNGStep:=9991;	
																END_IF;
													ELSIF CA_CarryingPos1  THEN//负极在取片位	
                                                                  DTPosError[12]:=FALSE;																	
																IF arrAxisCtrl[AxiseNo.AxisName.SEPTATLine].Cmd.arrbRealPoint[2]  THEN
																	DT_SingeMode();//单步选择										
																	An_OverNGStep:=1300;//
																ELSIF arrAxisCtrl[AxiseNo.AxisName.SEPTATLine].Cmd.arrbRealPoint[1] THEN
																	DT_SingeMode();//单步选择										
																	An_OverNGStep:=1400;//
																ELSE
																	Mach_Control.DT_b.Error[6]:=TRUE;//叠正极片凸轮耦合时，隔膜平移轴即不在正极叠片位，也不在正极叠片位报警
																	//An_OverNGStep:=9992;	
																END_IF;							
													ELSIF Scan_TON[1].Q THEN
																Scan_TON[1].IN:=FALSE;	
																//An_OverNGStep:=9993;
															   DTPosError[12]:=TRUE;
													END_IF
							    	ELSE
											IF (Ca_Step0=0 OR Ca_Step0=6666) AND (Ca_Step3=0 OR Ca_Step3=6666) AND Scan_TON[2].Q THEN
												Scan_TON[2].IN:=FALSE;		
												//An_OverNGStep:=9994;
												DTPosError[11]:=TRUE;
											END_IF
								END_IF
					END_IF		

              1600:	 //正极叠片升降移动至放片高度 		  
	           			IF NOT DP_SinStepe THEN					
									 IF arrAxisCtrl[AxiseNo.AxisName.AnDTCarryingUpDown].Status.Homed AND arrAxisCtrl[AxiseNo.AxisName.AnDTCarryingUpDown].Status.NoMoving AND 
										NOT arrAxisCtrl[AxiseNo.AxisName.AnDTCarryingUpDown].Status.Error AND arrAxisCtrl[AxiseNo.AxisName.AnDTCarryingLine].Cmd.arrbRealPoint[2] AND
                                             arrAxisCtrl[AxiseNo.AxisName.LeftYDUpDown].Cmd.arrbRealPoint[1] AND arrAxisCtrl[AxiseNo.AxisName.RightYDUpDown].Cmd.arrbRealPoint[1]       THEN
											IF arrAxisCtrl[AxiseNo.AxisName.AnDTCarryingUpDown].Cmd.arrbRealPoint[3] THEN
												arrAxisCtrl[AxiseNo.AxisName.AnDTCarryingUpDown].Cmd.iGoSetPos:=0;
											ELSE
												arrAxisCtrl[AxiseNo.AxisName.AnDTCarryingUpDown].Cmd.iGoSetPos:=3;//正极叠片升降移动至等待高度
											END_IF
									END_IF   	
								IF arrAxisCtrl[AxiseNo.AxisName.AnDTCarryingUpDown].Cmd.arrbRealPoint[3] THEN
								    DT_SingeMode();//单步选择
									An_OverNGStep:=1610;
								END_IF		
                       END_IF	   
		1610://	右刀升降轴上升至张开高度
						     arrCyCtrl[arrCyNo.ElectValveName.AnDTCarryingVacuum].Cmd.bOFF:=TRUE;//正极叠片搬运升降真空开
	                    	arrCyCtrl[arrCyNo.ElectValveName.AnDTCarryingVacuum].Cmd.bON:=FALSE;//正极叠片搬运升降真空开
						IF NOT DP_SinStepe THEN								
								IF 	arrAxisCtrl[AxiseNo.AxisName.RightYDUpDown].Status.Homed AND arrAxisCtrl[AxiseNo.AxisName.RightYDUpDown].Status.NoMoving THEN
									IF arrAxisCtrl[AxiseNo.AxisName.RightYDUpDown].Cmd.arrbRealPoint[15] THEN
										arrAxisCtrl[AxiseNo.AxisName.RightYDUpDown].Cmd.iGoSetPos:=0;
									ELSE
										arrAxisCtrl[AxiseNo.AxisName.RightYDUpDown].Cmd.iGoSetPos:=15;//右压刀升降上升至抽刀高度
									END_IF
								END_IF				
								IF arrAxisCtrl[AxiseNo.AxisName.RightYDUpDown].Cmd.arrbRealPoint[15] THEN
							     	DT_SingeMode();//单步选择
									An_OverNGStep:=1620;
								END_IF
						END_IF	   
	
            1620://	右压刀开合轴至张开位			   
					   IF NOT DP_SinStepe THEN
										IF 	arrAxisCtrl[AxiseNo.AxisName.RightYDLine].Status.Homed AND arrAxisCtrl[AxiseNo.AxisName.RightYDLine].Status.NoMoving THEN
												IF arrAxisCtrl[AxiseNo.AxisName.RightYDLine].Cmd.arrbRealPoint[2] THEN
													arrAxisCtrl[AxiseNo.AxisName.RightYDLine].Cmd.iGoSetPos:=0;
												ELSE
													arrAxisCtrl[AxiseNo.AxisName.RightYDLine].Cmd.iGoSetPos:=2;//右压刀开合至张开位	
												END_IF		
										END_IF;	
											IF arrAxisCtrl[AxiseNo.AxisName.RightYDLine].Cmd.arrbRealPoint[2] THEN
													DT_SingeMode();//单步选择
													An_OverNGStep:=1630;											
											END_IF
							END_IF;
				   
	
